Omron CX-Programmer project NewProject (CX-Programmer 9.32)

# PLC NewPLC1: CP1H XA

## Global symbols (name address type ; comment)
AGITATOR SCP
0.00 BOOL  ; Tablet Countinng Proxy
0.01 BOOL  ; Air pressure
0.02 BOOL  ; Turret Motor Overload
0.03 BOOL  ; LH Feeder Motor Overload
0.04 BOOL  ; LH Tamping
0.05 BOOL  ; RH Dozzer Asembly
0.06 BOOL  ; LH Main Set Pressure
0.07 BOOL  ; RH Tamping
0.08 BOOL  ; Guards Limit Switch
0.09 BOOL  ; LH Dozzer Assembly
0.10 BOOL  ; Std. Lubrication Oil Level Low
0.11 BOOL  ; Hydraulic Pressure S/w
100.00 BOOL  ; Main Motor
100.01 BOOL  ; Agitator Motor
100.02 BOOL  ; LH Feeder Motor
100.03 BOOL  ; RH Feeder Motor
100.04 BOOL  ; Hyd. Motor
100.05 BOOL  ; Sampling Gate
100.06 BOOL  ; Hyd. Dec SOV
100.07 BOOL  ; Magnetic Clutch
101.00 BOOL  ; 1 st Layer Sampling Gate ON
101.01 BOOL  ; 1 st Layer Sampling Gate OFF
101.02 BOOL  ; Lubrication Sol. On
101.03 BOOL  ; Comp. Zone Light
101.04 BOOL  ; Dust Extractor
101.05 BOOL  ; LPSL SOV
101.06 BOOL  ; Sampling Hooter
101.07 BOOL  ; Hooter
102 CHANNEL  ; RH Feeder Speed Reference
106.00 BOOL  ; LH Discharge SOV
106.01 BOOL  ; LH Filteration SOV
106.02 BOOL  ; LH Conveyour SOV
106.03 BOOL  ; RH Discharge SOV
106.04 BOOL  ; RH Filteration SOV
106.05 BOOL  ; RH Conveyour SOV
106.06 BOOL  ; Vacuum Pump
1.00 BOOL  ; RH Main Set Pressure
1.01 BOOL  ; RH Feeder Motor Overload
1.02 BOOL  ; Hyd. Motor O/L
1.03 BOOL  ; Emergency Stop
1.04 BOOL  ; LH Powder Level Low
1.05 BOOL  ; RH Powder Level Low
1.06 BOOL  ; Hyd. Oil Level Low
1.07 BOOL  ; LH Feeder Jamming
1.08 BOOL  ; RH Feeder Jamming
1.09 BOOL  ; Door For Ele. Panel Box
1.10 BOOL  ; Hand Wheel Guard
1.11 BOOL  ; Agitator Motor O/L
200 CHANNEL  ; Spare
201 CHANNEL  ; Turret Motor Current
2012 CHANNEL  ; LH Main Punch Force Input
202 CHANNEL  ; Hyd. System Pressure (4-20mA)
203 CHANNEL  ; Spare
210 CHANNEL  ; Turret Motor Speed Reference
211 CHANNEL  ; LH Feeder RPM Speed Refence
2.00 BOOL  ; LOWER GUARD LH OPEN
2.01 BOOL  ; $?St$Bk?_#[591] / LOWER GUARD RH OPEN / $?St$Bk?_#[591]
2.02 BOOL  ; UPPER GUARD FRONT OPEN
2.03 BOOL  ; UPPER GUARD LH OPEN
2.04 BOOL  ; UPPER GUARD RH OPEN
2.05 BOOL  ; UPPER GUARD REAR OPEN
2.06 BOOL  ; Int. Lub Motor Overload/LH POWDER LEVEL VERY LOW
2.07 BOOL  ; Int. Lub Oil Level Low/RH POWDER LEVEL VERY LOW
3.00 BOOL  ; Vacuum Pump O/L
3.01 BOOL  ; Vacum Pump Run Feedback
3.02 BOOL  ; LH Hopper Level High
3.03 BOOL  ; RH Hopper Level High
3.04 BOOL  ; Phase Failure
60 CHANNEL  ; minutes
A351 CHANNEL  ; MINUTE & SECOND
A352 CHANNEL  ; DATE & HOUR
A353 CHANNEL  ; YEAR & MONTH
C0 CHANNEL  ; Turret RPM Counter
C0001 BOOL  ; Lubrication ON Time
C0002 BOOL  ; Lubrication OFF Time
C0003 BOOL  ; Tablet Counter C3
C0005 BOOL  ; Reject Tab. / Rev.
C0006 BOOL  ; High Rejection For 3 Rot.
C0007 BOOL  ; Punch Tight Counter
C0008 BOOL  ; Counter For Sample
C0009 BOOL  ; Counter For Intermittent Cycle
C0010 BOOL  ; Total Rej. In 1 Batch
C0012 BOOL  ; First Rot. Rej. Counter
C0020 BOOL  ; LPSL ON Time
C0021 BOOL  ; LPSL OFF Time
C0025 BOOL  ; second counting
C0026 BOOL  ; minute counting
C0027 BOOL  ; hour counting
C0030 BOOL  ; Sampling interval timer
C0031 BOOL  ; 5 Min delay for machine stop
C0051 BOOL  ; LH Level High CNT
C0052 BOOL  ; RH Level High CNT
C0053 BOOL  ; LH Discharge CNT
C0054 BOOL  ; LH Delay CNT
C0055 BOOL  ; LH Filteration CNT
C0056 BOOL  ; LH Conv CNT
C0057 BOOL  ; RH Discharge CNT
C0058 BOOL  ; RH Delay CNT
C0059 BOOL  ; RH Filteration CNT
C0060 BOOL  ; RH Conv CNT
C11 CHANNEL  ; Total Sample Tab. In 1 Batch
D0 CHANNEL  ; Actual Screen
D1 CHANNEL  ; Operator Password
D1000 CHANNEL  ; Total Tablet Produced LSB
D1005 CHANNEL  ; Total Tablet Produced MSB
D101 CHANNEL  ; Actual Turret RPM
D1050 CHANNEL  ; Total Tablet Produced
D109 CHANNEL  ; Total Tablet Produced Higher Bit
D1100 CHANNEL  ; Main Force Data Range 1100-1199
D1110 CHANNEL  ; Actual Batch size
D1114 CHANNEL  ; Current Range
D116 CHANNEL  ; Current Factor (Count)
D122 CHANNEL  ; Turret Motor Current
D123 CHANNEL  ; Set Lubrication ON Time (Sec.)
D124 CHANNEL  ; Set Lubrication OFF Time (Min.)
D126 CHANNEL  ; Lubrication OFF Time (Min)
D127 CHANNEL  ; Actual Lub. ON Time
D128 CHANNEL  ; Actual Lub. OFF Time
D130 CHANNEL  ; Time For Punch Force Data
D135 CHANNEL  ; Time for Air Blow
D139 CHANNEL  ; Air Blow Delay Time
D141 CHANNEL  ; Air Blow Time Delay
D142 CHANNEL  ; Tablet Counting C3 Data
D152 CHANNEL  ; Main Force Data
D154 CHANNEL  ; High Rejection Limit
D155 CHANNEL  ; Low Rejection Limit
D156 CHANNEL  ; Main Force Data Count
D157 CHANNEL  ; Total Main Force
D159 CHANNEL  ; M/C Station
D161 CHANNEL  ; Main Avg. Force
D165 CHANNEL  ; Avg. Force For Die Fill PID Control
D173 CHANNEL  ; Punch Force For Graph
D180 CHANNEL  ; Force Rejection For Punch1
D181 CHANNEL  ; Force Rejection For Punch2
D182 CHANNEL  ; Force Rejection For Punch3
D183 CHANNEL  ; Force Rejection For Punch4
D184 CHANNEL  ; Force Rejection For Punch5
D185 CHANNEL  ; Air Blow ON Time
D186 CHANNEL  ; Air Blow ON Time (BCD)
D190 CHANNEL  ; Sample Punch No 1
D191 CHANNEL  ; Sample Punch No 2
D192 CHANNEL  ; Sample Punch No 3
D193 CHANNEL  ; Sample Punch No 4
D194 CHANNEL  ; Sample Punch No 5
D195 CHANNEL  ; Counter/Time Value For Sampling
D198 CHANNEL  ; Sample Time
D2 CHANNEL  ; Manager Password
D200 CHANNEL  ; minutes
D2000 CHANNEL  ; MINUTE & SECOND
D2002 CHANNEL  ; SEC
D2003 CHANNEL  ; MIN
D201 CHANNEL  ; hours
D2012 CHANNEL  ; HOUR
D2013 CHANNEL  ; DATE
D2022 CHANNEL  ; MONTH
D2023 CHANNEL  ; YEAR
D21 CHANNEL  ; Password for Login
D22 CHANNEL  ; Operator Password
D226 CHANNEL  ; Time Interval for Sampling (Sec)
D23 CHANNEL  ; Supervisor Password
D230 CHANNEL  ; Sampling Gate ON Time
D232 CHANNEL  ; Time For Intermittent Cycle
D236 CHANNEL  ; Total Rej. In 1 Batch
D238 CHANNEL  ; Total Sample Tab. In 1 Batch
D24 CHANNEL  ; Manager Password
D241 CHANNEL  ; High Force Control Limit
D242 CHANNEL  ; Low Force Control Limit
D243 CHANNEL  ; Initial Rejection Tablet
D245 CHANNEL  ; Enter Sync. Percentage
D25 CHANNEL  ; Selection Change Password
D250 CHANNEL  ; Vac-U-Max Control
D252 CHANNEL  ; (Set Turret RPM-Min RPM)
D254 CHANNEL  ; LH Delay Time
D256 CHANNEL  ; LH Filteration Time
D258 CHANNEL  ; Set Main Pressure
D26 CHANNEL  ; Enter Old Password
D260 CHANNEL  ; Set Tamping Pressure
D261 CHANNEL  ; Set Depth of Die Fill
D262 CHANNEL  ; Set Main Tablet Thickness
D264 CHANNEL  ; Set Tamp. Tab. Thickness
D266 CHANNEL  ; Actual Depth of Die Fill
D268 CHANNEL  ; Actual Tablet Thickness
D27 CHANNEL  ; Enter New Password
D270 CHANNEL  ; Actual Tamping Tablet Thickness
D272 CHANNEL  ; Main Upper Punch Entry
D274 CHANNEL  ; Tamping Upper Punch Entry
D275 CHANNEL  ; Message For Sampling collection
D276 CHANNEL  ; Die Fill Position message
D277 CHANNEL  ; Tablet Thickness Message
D278 CHANNEL  ; Tamp. Tablet Thickness Message
D28 CHANNEL  ; 0=Enter Password 1= Password OK 2=Invalid Password
D280 CHANNEL  ; RH Dischrge Time (BCD)
D286 CHANNEL  ; Tamping Force Data
D288 CHANNEL  ; LH High Level Disappear Time (BCD)
D29 CHANNEL  ; Change Password Message
D290 CHANNEL  ; RH High Level Disappear Time (BCD)
D296 CHANNEL  ; Total Cycle
D298 CHANNEL  ; Total Cycle (BCD)
D30 CHANNEL  ; RH Feeder RPM
D300 CHANNEL  ; RH Feeder RPM
D3015 CHANNEL  ; LH scp input min
D3016 CHANNEL  ; LH scp scal min
D3017 CHANNEL  ; LH scp scal max
D3018 CHANNEL  ; LH scp input max
D3019 CHANNEL  ; Actual LH Punch Force
D302 CHANNEL  ; Hour
D304 CHANNEL  ; Min
D306 CHANNEL  ; Sec
D319 CHANNEL  ; RH Store Feeder RPM
D330 CHANNEL  ; Sampling inteval time min
D3508 CHANNEL  ; Operator Code
D3509 CHANNEL  ; Recipe Code
D3525 CHANNEL  ; Batch Size
D360 CHANNEL  ; Tamp. Avg Force
D364 CHANNEL  ; Tamping Trend Graph
D368 CHANNEL  ; Avg. Ejection Data
D39 CHANNEL  ; RH Store Feeder RPM
D40 CHANNEL  ; Store Screen
D4000 CHANNEL  ; minutes
D4001 CHANNEL  ; hours
D406 CHANNEL  ; Ejection Force Data
D432 CHANNEL  ; Die Fill MIN
D433 CHANNEL  ; Die Fill MAX
D435 CHANNEL  ; Machine Station
D44 CHANNEL  ; Set Turret RPM (Store)
D480 CHANNEL  ; Acceleration
D481 CHANNEL  ; Deacceleration
D482 CHANNEL  ; Frequency
D484 CHANNEL  ; Pulses
D486 CHANNEL  ; Start Frequency
D499 CHANNEL  ; Main Lower Punch Position
D500 CHANNEL  ; Tamping interlock
D501 CHANNEL  ; Main Pressure Interlock
D510 CHANNEL  ; Set LPSL ON Time
D511 CHANNEL  ; Set LPSL OFF Time
D512 CHANNEL  ; LPSL ON TIME (Sec)
D513 CHANNEL  ; LPSL OFF TIME (Min)
D514 CHANNEL  ; Output Pulse to be Generate
D515 CHANNEL  ; Act. LPSL ON Time
D516 CHANNEL  ; Act. LPSL OFF Time
D52 CHANNEL  ; LH Set Feeder RPM
D520 CHANNEL  ; Hyd. Low Limit
D521 CHANNEL  ; Hyd. High Limit
D522 CHANNEL  ; Hyd. Limit Low (Comp)
D523 CHANNEL  ; Hyd. Limit High (Comp)
D525 CHANNEL  ; Hyd. Sys. Pr. Message
D527 CHANNEL  ; Act. Hyd. Pressure
D528 CHANNEL  ; Hyd. Graph
D53 CHANNEL  ; LH Store Feeder RPM
D530 CHANNEL  ; SCL_P
D533 CHANNEL  ; SCL_P3
D535 CHANNEL  ; Total travel in mm/100
D539 CHANNEL  ; Tamping Lower Punch Position
D54 CHANNEL  ; LH Store Feeder RPM
D542 CHANNEL  ; Total Cup Depth
D548 CHANNEL  ; Lower punch pos + Total Cup Depth
D550 CHANNEL  ; Set Agitator RPM
D552 CHANNEL  ; Act Agitiator RPM
D56 CHANNEL  ; Feeder RPM (Float)
D572 CHANNEL  ; Time Interval For Sampling (BCD) - Sec
D578 CHANNEL  ; Die Fill High+Low Limit
D579 CHANNEL  ; Die Fill High/Low Avg Limit
D60 CHANNEL  ; RH Feeder O/P
D601 CHANNEL  ; Set Main  + Relief
D602 CHANNEL  ; Set Tamping + Relief Value
D606 CHANNEL  ; No of Tablet Counter
D615 CHANNEL  ; Min. Main Force
D6150 CHANNEL  ; -
D6152 CHANNEL  ; Total Rejec.+Sample Tab
D6158 CHANNEL  ; Powder Delay Time
D6160 CHANNEL  ; M/c Stn (Print)
D6168 CHANNEL  ; Feeder Post Run Time (BCD)
D617 CHANNEL  ; Max. Main Force
D619 CHANNEL  ; Min. Tamp. Force
D621 CHANNEL  ; Max. Tamp. Force
D64 CHANNEL  ; Scale Min
D66 CHANNEL  ; Scale Range
D67 CHANNEL  ; \
D7 CHANNEL  ; '
D70 CHANNEL  ; Die Fill Position
D700 CHANNEL  ; Lower Punch position at last time
D7005 CHANNEL  ; Batch Size
D702 CHANNEL  ; Store lower punch Position at last time
D7050 CHANNEL  ; Hour
D7052 CHANNEL  ; Min
D7060 CHANNEL  ; Sample + Reject Tab
D7064 CHANNEL  ; Good Tablet
D707 CHANNEL  ; Generate Pulse at last time
D709 CHANNEL  ; Total Travel at last time
D710 CHANNEL  ; Required pulse for travel at last time
D712 CHANNEL  ; Overl pulse at last time
D715 CHANNEL  ; Pulse feedback
D720 CHANNEL  ; Every 0.2 sec Set Tamp. Tab Thickness
D74 CHANNEL  ; LH Actual Feeder RPM
D746 CHANNEL  ; Powder Feeding Selection
D747 CHANNEL  ; Hour Meter 0:Reset 1:Start
D748 CHANNEL  ; Guard Interlock
D749 CHANNEL  ; Dummy Selection
D75 CHANNEL  ; Set Turret RPM
D750 CHANNEL  ; Dummy 1
D751 CHANNEL  ; Dummy 2
D752 CHANNEL  ; Dummy 3
D753 CHANNEL  ; Dummy 4
D754 CHANNEL  ; Dummy 5
D756 CHANNEL  ; Mode of Sampling
D758 CHANNEL  ; Compaction Mode 0: Manual 1: Auto
D759 CHANNEL  ; SCADA_BYPASS
D76 CHANNEL  ; Store Turret RPM
D762 CHANNEL  ; Dummy Punch Count
D764 CHANNEL  ; Total Dummy Punch
D766 CHANNEL  ; Final Total Punch
D768 CHANNEL  ; Tab w Dummy Punch
D77 CHANNEL  ; RH Actual Feeder RPM
D78 CHANNEL  ; RPM (Float)
D8 CHANNEL  ; Change Screen
D800 CHANNEL  ; Act. Hyd. Pressure Print
D82 CHANNEL  ; Input Max
D86 CHANNEL  ; Scale Min
D88 CHANNEL  ; Scale Range
D96 CHANNEL  ; Used for Turret RPM Calculation
D99 CHANNEL  ; Total No. Of Punch
H100.00 BOOL  ; Dummy Punch Selection
H100.01 BOOL  ; 0: Gravity 1: Force Feeder
H100.02 BOOL  ; Sampling ON/OFF
H100.03 BOOL  ; Batch Reseted
H101 CHANNEL  ; Hydrualic Pressure
H101.00 BOOL  ; Lub, Healthy
H102 CHANNEL  ; Hydraulic Pressure for Graph
H102.00 BOOL  ; LPSL ON Time : Low Limit
H102.01 BOOL  ; LPSL ON Time : Upper Limit
H102.02 BOOL  ; LPSL OFF Time : Low Limit
H102.03 BOOL  ; LPSL OFF Time : Upper Limit
H102.04 BOOL  ; LPSL Healthy
H102.05 BOOL  ; 1 Min Pulse
H103 CHANNEL  ; Turret Motor Current * 10
H103.00 BOOL  ; System Pr. High IL
H103.01 BOOL  ; Sys. Pr. Low IL
H103.02 BOOL  ; Hyd. Sys. Pr. High
H103.03 BOOL  ; Hyd. Sys. Pr. Low
H103.05 BOOL  ; 0: Hyd. Manual 1: Hyd. Auto
H103.06 BOOL  ; Hyd. Healthy
H103.07 BOOL  ; Hyd. INC
H103.08 BOOL  ; Hyd. DEC
H103.15 BOOL  ; All Upper Punch Free
H105.00 BOOL  ; Scada 0: OFF 1:Running
H105.01 BOOL  ; Scada 0: Bypass 1: Interlock
H107 CHANNEL  ; Actual Tab/Min
H10.00 BOOL  ; Bilayer sel. 1: standard 0: Bilayer
H10.01 BOOL  ; Bilayer Sampling
H10.02 BOOL  ; Calibration bit for current in calibration screen
H10.04 BOOL  ; Bilayer Sampling ON
H10.05 BOOL  ; Bilayer sampled on
H110.00 BOOL  ; Punch Tight 1
H110.01 BOOL  ; Punch Tight 2
H110.02 BOOL  ; Punch Tight 3
H110.03 BOOL  ; Punch Tight 4
H110.04 BOOL  ; Punch Tight 5
H110.05 BOOL  ; Punch Tight 6
H110.06 BOOL  ; Punch Tight 7
H110.07 BOOL  ; Punch Tight 8
H110.08 BOOL  ; Punch Tight 9
H110.09 BOOL  ; Punch Tight 10
H110.10 BOOL  ; Punch Tight 11
H110.11 BOOL  ; Punch Tight 12
H110.12 BOOL  ; Punch Tight 13
H110.13 BOOL  ; Punch Tight 14
H110.14 BOOL  ; Punch Tight 15
H110.15 BOOL  ; Punch Tight 16
H111.00 BOOL  ; Punch Tight 17
H111.01 BOOL  ; Punch Tight 18
H111.02 BOOL  ; Punch Tight 19
H111.03 BOOL  ; Punch Tight 20
H111.04 BOOL  ; Punch Tight 21
H111.05 BOOL  ; Punch Tight 22
H111.06 BOOL  ; Punch Tight 23
H111.07 BOOL  ; Punch Tight 24
H111.08 BOOL  ; Punch Tight 25
H111.09 BOOL  ; Punch Tight 26
H111.10 BOOL  ; Punch Tight 27
H111.11 BOOL  ; Punch Tight 28
H111.12 BOOL  ; Punch Tight 29
H111.13 BOOL  ; Punch Tight 30
H111.14 BOOL  ; Punch Tight 31
H111.15 BOOL  ; Punch Tight 32
H112.00 BOOL  ; Punch Tight 33
H112.01 BOOL  ; Punch Tight 34
H112.02 BOOL  ; Punch Tight 35
H112.03 BOOL  ; Punch Tight 36
H112.04 BOOL  ; Punch Tight 37
H118 CHANNEL  ; Actual Turret RPM
H11.00 BOOL  ; Download Recipe
H11.01 BOOL  ; Bilayer Sampling latch bit
H123 CHANNEL  ; Batch Recipe Code
H12.14 BOOL  ; Screen Move for MS1
H12.15 BOOL  ; Screen Move for MS2
H140.00 BOOL  ; Agitator Jog
H140.01 BOOL  ; Agitator ON/OFF
H150 CHANNEL  ; Total Tablet Produced Lower Bit
H150.01 BOOL  ; View Recipe
H150.02 BOOL  ; Download Recipe
H150.03 BOOL  ; Batch Print
H150.04 BOOL  ; Batch Print ON
H150.05 BOOL  ; Batch Start (Once)
H151.00 BOOL  ; MS1 Screen
H151.01 BOOL  ; MS2 SCREEN
H151.02 BOOL  ; Auto Return From MS1
H151.03 BOOL  ; Return
H151.04 BOOL  ; Auto Return From MS2
H151.05 BOOL  ; Auto Return From MS3
H151.06 BOOL  ; MS3 screen
H151.07 BOOL  ; MS4 screen
H151.08 BOOL  ; Auto Return From MS4
H16.00 BOOL  ; Sampling Alarm Time cycle Latch
H16.01 BOOL  ; Sampling timer Done
H16.02 BOOL  ; 5 Min delay timer done
H16.04 BOOL  ; Hooter on
H17.00 BOOL  ; Interlock for Sampling time Inc
H17.01 BOOL  ; Interlock for Sampling time Dec
H18.00 BOOL  ; Dust Ext. Start
H18.01 BOOL  ; Dust Ext. Stop
H18.02 BOOL  ; Dust Ext. On
H21.00 BOOL  ; Operator
H21.01 BOOL  ; Supervisor
H21.02 BOOL  ; Manager
H21.08 BOOL  ; Supervisor / Manger Login
H21.09 BOOL  ; Operator Password OK
H21.10 BOOL  ; Supervisor Password OK
H21.11 BOOL  ; Manager Password OK
H21.12 BOOL  ; Password OK
H222.00 BOOL  ; Batch Complete Latch
H22.00 BOOL  ; Operator Old Password OK
H22.01 BOOL  ; Supervisor Old Password OK
H22.02 BOOL  ; Manager Old Password OK
H22.03 BOOL  ; Old Password OK
H22.05 BOOL  ; Security Control Bit
H22.06 BOOL  ; Master Password Bit
H22.07 BOOL  ; Operator Once Bit
H22.08 BOOL  ; Supervisor Once Bit
H22.09 BOOL  ; Manager Once Bit
H22.12 BOOL  ; Change Operator Password
H22.13 BOOL  ; Change Supervisor Password
H22.14 BOOL  ; Change Manager Password
H23.01 BOOL  ; Change Operator Password Once Bit
H23.03 BOOL  ; Change Supervisor Password Once Bit
H23.05 BOOL  ; Change Manager Password Once Bit
H25.01 BOOL  ; Air Pressure Set
H25.07 BOOL  ; Int Lub oil Level Low Latch
H25.10 BOOL  ; Lubrication Oil Level Low Set
H25.11 BOOL  ; Hydraulic Pressure S/w Set
H26.06 BOOL  ; Hyd. Oil Level Low Set
H36.00 BOOL  ; Vac-U-Max Reset
H36.01 BOOL  ; Vac-U-Max Start/Stop
H36.02 BOOL  ; Vac-U-Max Hault
H36.05 BOOL  ; Vac-U-Max Healthy Auto
H36.06 BOOL  ; LH Vac-U-Max Running
H36.07 BOOL  ; RH Vac-U-Max Running
H36.08 BOOL  ; Total Cycle Complete
H36.09 BOOL  ; LH Hopper Level High (Latch)
H36.10 BOOL  ; RH Hopper Level High (Latch)
H387 CHANNEL  ; h120
H400.00 BOOL  ; Hooter Reset
H400.05 BOOL  ; Hooter latch
H50.00 BOOL  ; VAC U MAX 0=man 1=auto
H50.01 BOOL  ; LH Discharge SOV ON/OFF
H50.02 BOOL  ; LH Filteration SOV ON/OFF
H50.03 BOOL  ; LH Conveyour SOV ON/OFF
H50.04 BOOL  ; RH Discharge SOV ON/OFF
H50.05 BOOL  ; RH Filteration SOV ON/OFF
H50.06 BOOL  ; RH Conveyour SOV ON/OFF
H50.07 BOOL  ; Vacuum Pump ON/OFF
H51.00 BOOL  ; Main Interlock Healthy
H51.01 BOOL  ; Main Motor Start
H51.02 BOOL  ; Main Motor RUN (Auto)
H51.03 BOOL  ; Main Motor Stop
H51.04 BOOL  ; Lubrication Jog
H51.05 BOOL  ; Turret & Feeder Jog
H51.06 BOOL  ; Clutch Engage
H51.07 BOOL  ; Clutch Latch
H51.08 BOOL  ; 0=Gurds Bypass 1=Guards Interlock
H51.09 BOOL  ; Clutch Disengage
H51.10 BOOL  ; 0=Manual 1=Auto
H51.11 BOOL  ; Lub.: 0=Auto 1= Manual
H51.12 BOOL  ; Turret Jog
H51.13 BOOL  ; LH Feeder Motor Jog
H51.14 BOOL  ; RH Feeder Motor Jog
H51.15 BOOL  ; Hydraulic Pressure Dec.
H52.01 BOOL  ; Rising Edge of Proxy
H52.04 BOOL  ; Interlock for Turret RPM Inc
H52.05 BOOL  ; Interlock for Turret RPM Dec
H52.06 BOOL  ; LH Interlock for Feeder RPM Inc
H52.07 BOOL  ; LH Interlock for Feeder RPM Dec
H52.08 BOOL  ; RH Interlock for Feeder RPM Inc
H52.09 BOOL  ; RH Interlock for Feeder RPM Dec
H52.10 BOOL  ; Main Motor (Test RUN)
H52.11 BOOL  ; LPSL 0: Manual 1: Auto
H52.12 BOOL  ; Initial Rej. Gate Dignostic
H52.13 BOOL  ; LPSL Jog
H53.00 BOOL  ; Batch Complete
H53.01 BOOL  ; Batch Reset
H53.02 BOOL  ; Lower Limit Lubrication ON Time
H53.03 BOOL  ; Upper Limit Lubrication ON Time
H53.04 BOOL  ; Lower Limit Lubrication OFF Time
H53.05 BOOL  ; Upper Limit Lubrication OFF Time
H53.07 BOOL  ; Interlock for Download
H53.07 BOOL  ; Access Denied
H53.08 BOOL  ; Print Command to Scada
H53.09 BOOL  ; Home Proxy not Proper
H53.10 BOOL  ; Tablet Count Proxy Not Proper
H53.12 BOOL  ; Die Fill at Min Limit
H53.13 BOOL  ; Die Fill at Max Limit
H54.00 BOOL  ; Selected Punch
H54.01 BOOL  ; All Tab. Continuous
H54.02 BOOL  ; All Tablet Intermittent
H54.03 BOOL  ; Dynemic Reject on
H54.04 BOOL  ; For 1 Rot. High Rejection
H54.05 BOOL  ; Tablet Rejection/Rev.
H54.06 BOOL  ; Counter NEQ Zero
H54.07 BOOL  ; No. of Tablet
H54.08 BOOL  ; Stop Reason Latch
H54.09 BOOL  ; Final Bit For Rej./Samp.
H54.10 BOOL  ; Air Blow ON Time Bit
H54.11 BOOL  ; Sample Enable For 1 Rot.
H54.12 BOOL  ; Rej. Air Blow On Dignostic
H54.13 BOOL  ; $?St$Bk?_#[592] / 0=Rotation 1=Time / (Now only Based on Time)$?St$Bk?_#[592]
H54.14 BOOL  ; 0=Sample OFF 1=Sample On
H54.15 BOOL  ; All Tablet Intermittent
H55 CHANNEL  ; Interlock Status
H55.00 BOOL  ; For Input Interlocks
H56 CHANNEL  ; Interlock Status
H56.00 BOOL  ; For Input Interlocks
H56 CHANNEL  ; Interlock Status
H57 CHANNEL  ; Interlock Status
H57.02 BOOL  ; LH POWDER VACCUM HOPPER
H57.03 BOOL  ; RH POWDER VACCUM HOPPER
H58.00 BOOL  ; Pop up for Access Denied
H59.01 BOOL  ; Sampleing Enable Bit
H59.02 BOOL  ; Reset for C8
H59.03 BOOL  ; Reset For C8 & C9
H59.04 BOOL  ; Complete Intermittent Cycle
H60.01 BOOL  ; Rejection/Sampling For Perticular Punch
H61.01 BOOL  ; Tab. For Sampling
H62.00 BOOL  ; 0=Sync. Manual 1=Sync. Auto
H62.01 BOOL  ; Main Pressure O/L
H62.02 BOOL  ; Tamping Pressure O/L
H62.03 BOOL  ; 0=Die Fill Manual 1= Diefill Auto
H62.04 BOOL  ; Die Fill  Maximum
H62.05 BOOL  ; Die Fill Minimum
H62.06 BOOL  ; Tablet Thickness Maximum
H62.07 BOOL  ; Tablet Thickness Minimum
H62.08 BOOL  ; Tamp. Tab. Thickness Maximum
H62.09 BOOL  ; Tamp. Tab. Thickness Minimum
H63.04 BOOL  ; Batch Start for Scada
H63.05 BOOL  ; Batch Complete for Scada
H64.00 BOOL  ; Avg Force < Lower Force Limit
H64.02 BOOL  ; Avg Force > Upper Force Limit
H64.04 BOOL  ; Die Fill Inc
H64.05 BOOL  ; Die Fill Dec
H64.06 BOOL  ; Die Fill INC (HMI)
H64.07 BOOL  ; Die Fill DEC (HMI)
H64.08 BOOL  ; Tamp. Tab Thickness Inc
H64.09 BOOL  ; Tamp. Tab. Thickness Dec.
H65.00 BOOL  ; Output Interlocks
H66.00 BOOL  ; Output Interlocks
H67.00 BOOL  ; Output Interlocks
H68.00 BOOL  ; Tamping Tablet Thickness Sevo Interlock
H68.01 BOOL  ; Tamping Servo REV at last time
H68.02 BOOL  ; Tamping servo FWD at Last time
H70.00 BOOL  ; 1 sec pulse o/p latch
H70.03 BOOL  ; All Tab. Cont.
H70.05 BOOL  ; No. of. Tab. Enb.
H70.07 BOOL  ; Ejection Force Limit Max
H70.10 BOOL  ; Batch No Enter
H72.05 BOOL  ; Vac U Max Healthy Man
H75.02 BOOL  ; Station 20
H75.03 BOOL  ; Station 24
H75.04 BOOL  ; Station 30
H77.00 BOOL  ; Agitator Interlock/Bypass
H77.14 BOOL  ; Reset all counter for RH & count 1 cycle
H77.15 BOOL  ; Reset all counter for LH & count 1 cycle
H7.01 BOOL  ; Manual Interlock
H7.02 BOOL  ; Test Turret Interlock
H7.03 BOOL  ; Test LH Feeder Interlock
H7.04 BOOL  ; Test RH Feeder Interlock
H7.05 BOOL  ; Test Air Interlock
H7.06 BOOL  ; Feeder Jaming 0: Bypass 1: Interlock
H7.07 BOOL  ; LH Feeder Jamming Interlock
H7.08 BOOL  ; RH Feeder Jamming Interlock
H80.00 BOOL  ; 0:Two Side,1:Single side
T0007 BOOL  ; Hyd. Dec SOV OFF Time
T0013 BOOL  ; LH Feeder Jamming Timer
T0018 BOOL  ; Sampling Gate ON Timer
T0023 BOOL  ; Clutch Engage (Aft Feeder Pre Run)
T0024 BOOL  ; Actual Pusle for every 10 Sec
T0025 BOOL  ; Clutch Delay (Auto)
T0028 BOOL  ; Feeder Post Run Timer
T0029 BOOL  ; Powder Level Timer
T0034 BOOL  ; LH Feeder RPM Actual Transfer Time
T0035 BOOL  ; Lubrication Automatically Auto after 5 Min.
T0036 BOOL  ; Access Denied Timer (1s)
T0037 BOOL  ; RH Feeder RPM Actual Transfer Time
HYD_PRESSURE SCP
Hyd_New SCP_Hyd
LH_FEEDER_SPEED SCP
RH_Feeder_Reference SCP
RTC_01 FRTC
Turret_Current SCP
Turret_Speed_reference SCP

## Program Main_Program (cyclic task 0)
Local symbols
AD0 CHANNEL
D441D454 CHANNEL
D441d454 CHANNEL
D442D452 CHANNEL
D444D454 CHANNEL
D4d425 INT
DD411 INT
Dd568 INT
Dd572 UINT_BCD
Dh102 INT
First_pass BOOL
P_0_01s BOOL
P_on BOOL  ; Always on flag
cf CHANNEL
cfg CHANNEL
ch0 CHANNEL
cio2 INT
cntr35 BOOL
ct4 BOOL
d INT
da CHANNEL
dx30 CHANNEL
end BOOL
h BOOL
ld700 UINT
out BOOL
p BOOL
p102 BOOL
p_1s BOOL  ; pulse for 1sec
p_ON BOOL
p_On BOOL
p_oFF BOOL
p_oN BOOL
p_on BOOL  ; always on flag
scl BOOL  ; d200
up BOOL
vw0 CHANNEL

### Section Password
; Pass Word

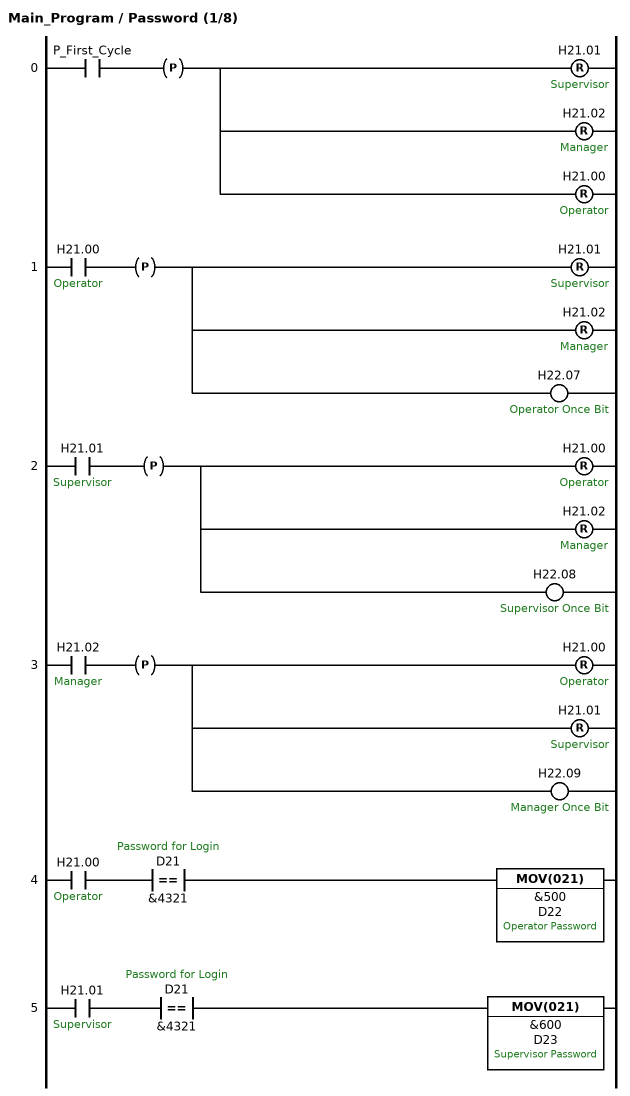
; rung 0
LD P_First_Cycle
UP(521)
RSET H21.01  ; Supervisor
RSET H21.02  ; Manager
RSET H21.00  ; Operator
; rung 1
LD H21.00  ; Operator
UP(521)
RSET H21.01  ; Supervisor
RSET H21.02  ; Manager
OUT H22.07  ; Operator Once Bit
; rung 2
LD H21.01  ; Supervisor
UP(521)
RSET H21.00  ; Operator
RSET H21.02  ; Manager
OUT H22.08  ; Supervisor Once Bit
; rung 3
LD H21.02  ; Manager
UP(521)
RSET H21.00  ; Operator
RSET H21.01  ; Supervisor
OUT H22.09  ; Manager Once Bit
; rung 4
LD H21.00  ; Operator
AND=(300) D21 &4321  ; Password for Login
MOV(021) &500 D22  ; Operator Password
; rung 5
LD H21.01  ; Supervisor
AND=(300) D21 &4321  ; Password for Login
MOV(021) &600 D23  ; Supervisor Password

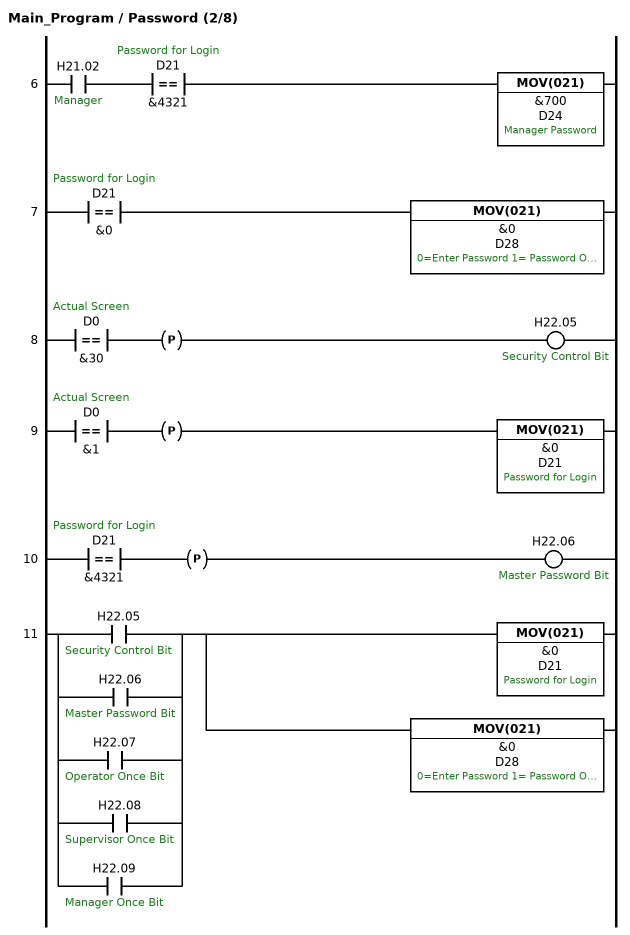
; rung 6
LD H21.02  ; Manager
AND=(300) D21 &4321  ; Password for Login
MOV(021) &700 D24  ; Manager Password
; rung 7
LD=(300) D21 &0  ; Password for Login
MOV(021) &0 D28  ; 0=Enter Password 1= Password OK 2=Invalid Password
; rung 8
LD=(300) D0 &30  ; Actual Screen
UP(521)
OUT H22.05  ; Security Control Bit
; rung 9
LD=(300) D0 &1  ; Actual Screen
UP(521)
MOV(021) &0 D21  ; Password for Login
; rung 10
LD=(300) D21 &4321  ; Password for Login
UP(521)
OUT H22.06  ; Master Password Bit
; rung 11
LD H22.05  ; Security Control Bit
OR H22.06  ; Master Password Bit
OR H22.07  ; Operator Once Bit
OR H22.08  ; Supervisor Once Bit
OR H22.09  ; Manager Once Bit
MOV(021) &0 D21  ; Password for Login
MOV(021) &0 D28  ; 0=Enter Password 1= Password OK 2=Invalid Password

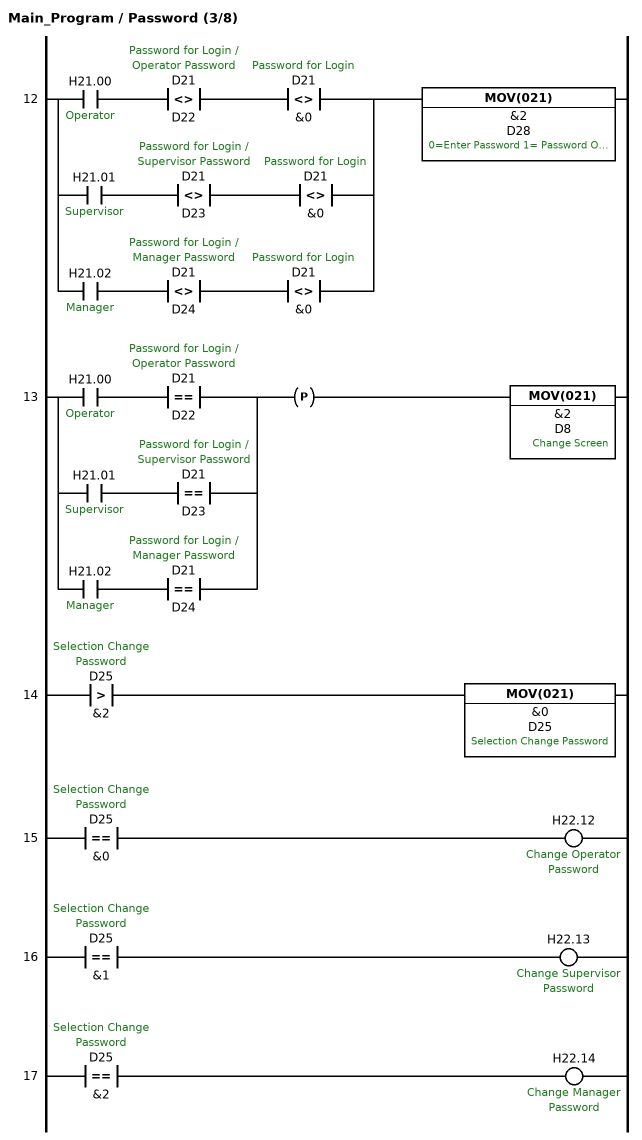
; rung 12
LD H21.00  ; Operator
AND<>(305) D21 D22  ; Password for Login, Operator Password
AND<>(305) D21 &0  ; Password for Login
LD H21.01  ; Supervisor
AND<>(305) D21 D23  ; Password for Login, Supervisor Password
AND<>(305) D21 &0  ; Password for Login
ORLD
LD H21.02  ; Manager
AND<>(305) D21 D24  ; Password for Login, Manager Password
AND<>(305) D21 &0  ; Password for Login
ORLD
MOV(021) &2 D28  ; 0=Enter Password 1= Password OK 2=Invalid Password
; rung 13
LD H21.00  ; Operator
AND=(300) D21 D22  ; Password for Login, Operator Password
LD H21.01  ; Supervisor
AND=(300) D21 D23  ; Password for Login, Supervisor Password
ORLD
LD H21.02  ; Manager
AND=(300) D21 D24  ; Password for Login, Manager Password
ORLD
UP(521)
MOV(021) &2 D8  ; Change Screen
; rung 14
LD>(320) D25 &2  ; Selection Change Password
MOV(021) &0 D25  ; Selection Change Password
; rung 15
LD=(300) D25 &0  ; Selection Change Password
OUT H22.12  ; Change Operator Password
; rung 16
LD=(300) D25 &1  ; Selection Change Password
OUT H22.13  ; Change Supervisor Password
; rung 17
LD=(300) D25 &2  ; Selection Change Password
OUT H22.14  ; Change Manager Password

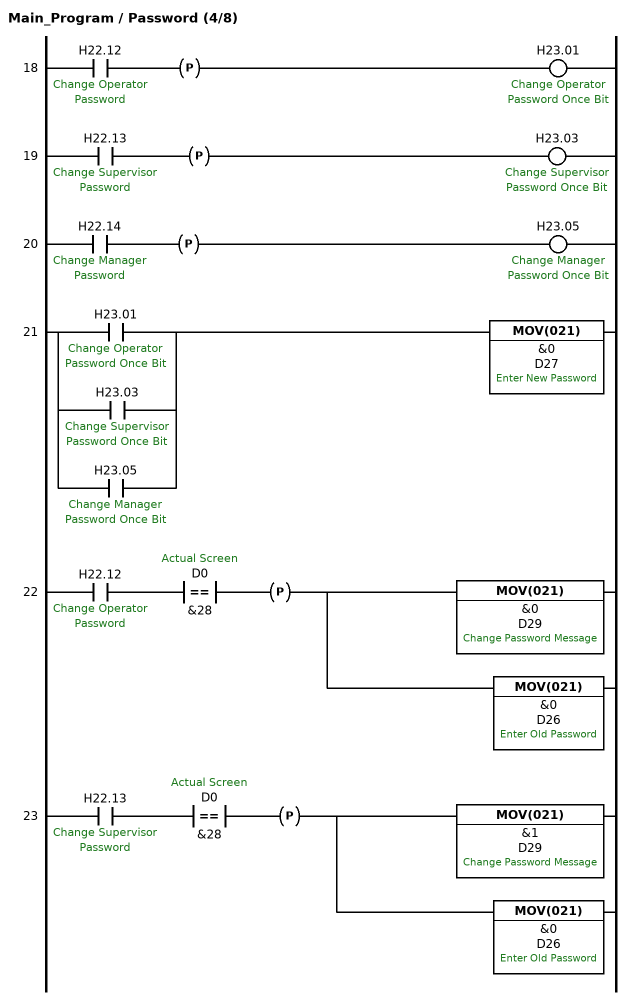
; rung 18
LD H22.12  ; Change Operator Password
UP(521)
OUT H23.01  ; Change Operator Password Once Bit
; rung 19
LD H22.13  ; Change Supervisor Password
UP(521)
OUT H23.03  ; Change Supervisor Password Once Bit
; rung 20
LD H22.14  ; Change Manager Password
UP(521)
OUT H23.05  ; Change Manager Password Once Bit
; rung 21
LD H23.01  ; Change Operator Password Once Bit
OR H23.03  ; Change Supervisor Password Once Bit
OR H23.05  ; Change Manager Password Once Bit
MOV(021) &0 D27  ; Enter New Password
; rung 22
LD H22.12  ; Change Operator Password
AND=(300) D0 &28  ; Actual Screen
UP(521)
MOV(021) &0 D29  ; Change Password Message
MOV(021) &0 D26  ; Enter Old Password
; rung 23
LD H22.13  ; Change Supervisor Password
AND=(300) D0 &28  ; Actual Screen
UP(521)
MOV(021) &1 D29  ; Change Password Message
MOV(021) &0 D26  ; Enter Old Password

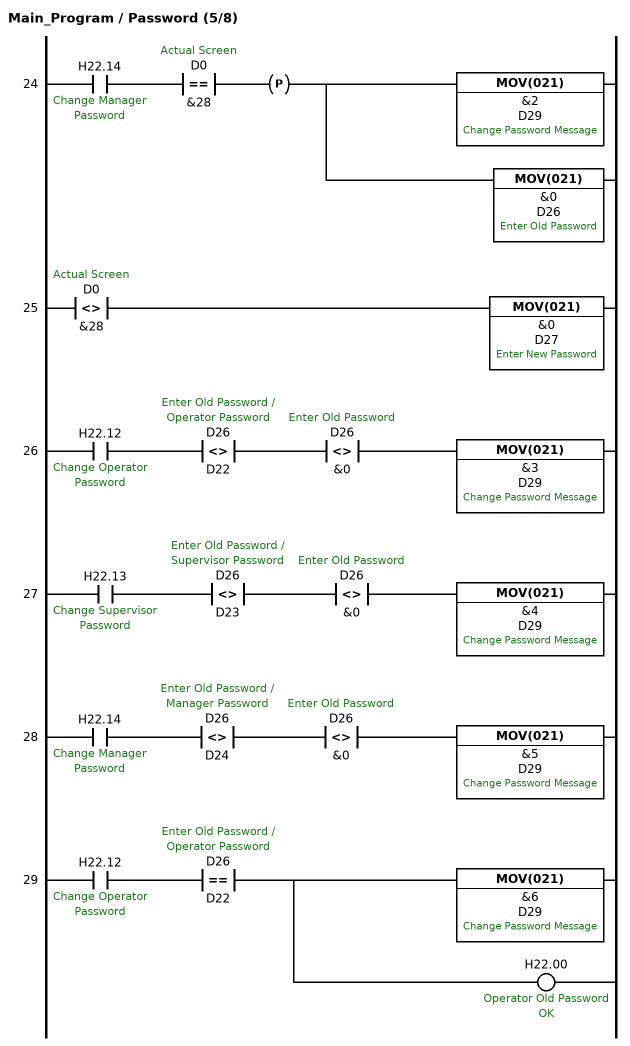
; rung 24
LD H22.14  ; Change Manager Password
AND=(300) D0 &28  ; Actual Screen
UP(521)
MOV(021) &2 D29  ; Change Password Message
MOV(021) &0 D26  ; Enter Old Password
; rung 25
LD<>(305) D0 &28  ; Actual Screen
MOV(021) &0 D27  ; Enter New Password
; rung 26
LD H22.12  ; Change Operator Password
AND<>(305) D26 D22  ; Enter Old Password, Operator Password
AND<>(305) D26 &0  ; Enter Old Password
MOV(021) &3 D29  ; Change Password Message
; rung 27
LD H22.13  ; Change Supervisor Password
AND<>(305) D26 D23  ; Enter Old Password, Supervisor Password
AND<>(305) D26 &0  ; Enter Old Password
MOV(021) &4 D29  ; Change Password Message
; rung 28
LD H22.14  ; Change Manager Password
AND<>(305) D26 D24  ; Enter Old Password, Manager Password
AND<>(305) D26 &0  ; Enter Old Password
MOV(021) &5 D29  ; Change Password Message
; rung 29
LD H22.12  ; Change Operator Password
AND=(300) D26 D22  ; Enter Old Password, Operator Password
MOV(021) &6 D29  ; Change Password Message
OUT H22.00  ; Operator Old Password OK

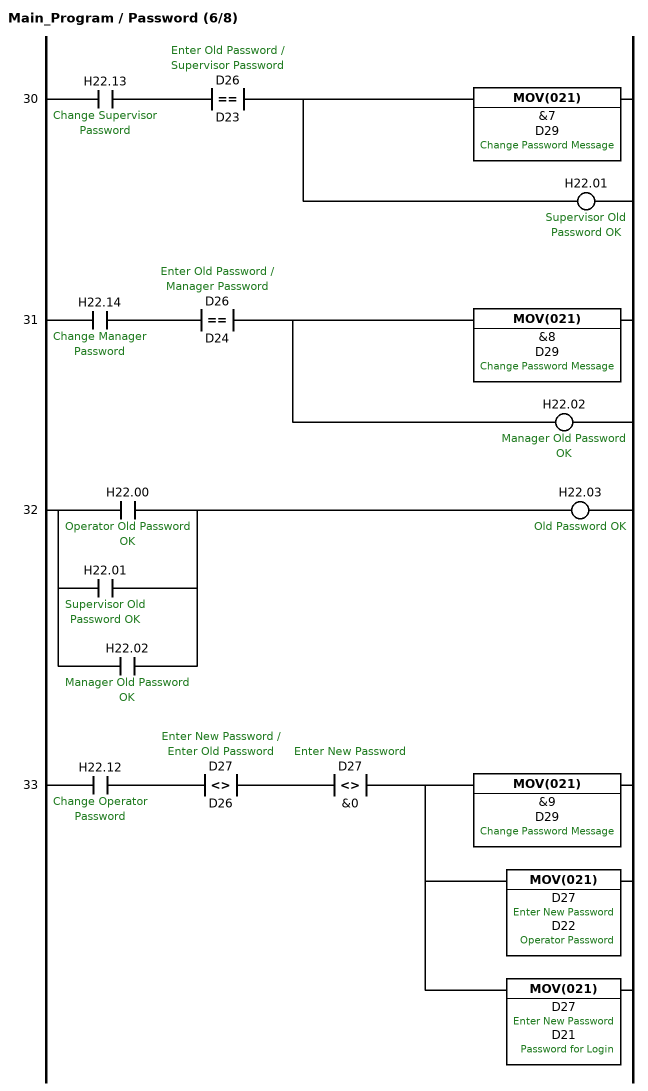
; rung 30
LD H22.13  ; Change Supervisor Password
AND=(300) D26 D23  ; Enter Old Password, Supervisor Password
MOV(021) &7 D29  ; Change Password Message
OUT H22.01  ; Supervisor Old Password OK
; rung 31
LD H22.14  ; Change Manager Password
AND=(300) D26 D24  ; Enter Old Password, Manager Password
MOV(021) &8 D29  ; Change Password Message
OUT H22.02  ; Manager Old Password OK
; rung 32
LD H22.00  ; Operator Old Password OK
OR H22.01  ; Supervisor Old Password OK
OR H22.02  ; Manager Old Password OK
OUT H22.03  ; Old Password OK
; rung 33
LD H22.12  ; Change Operator Password
AND<>(305) D27 D26  ; Enter New Password, Enter Old Password
AND<>(305) D27 &0  ; Enter New Password
MOV(021) &9 D29  ; Change Password Message
MOV(021) D27 D22  ; Enter New Password, Operator Password
MOV(021) D27 D21  ; Enter New Password, Password for Login

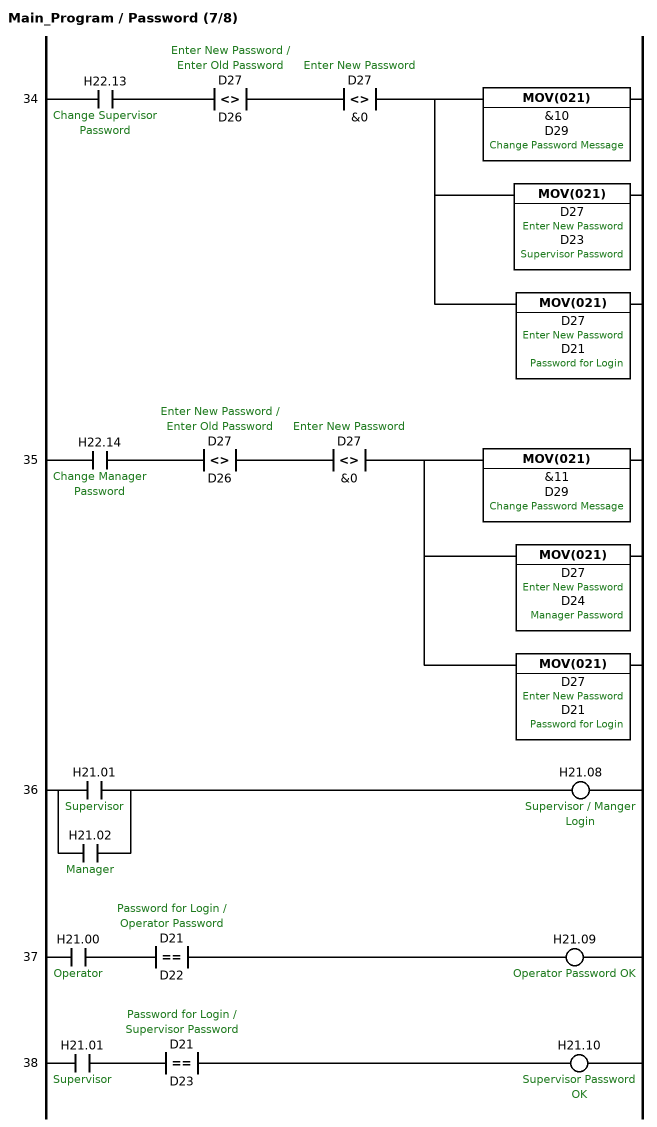
; rung 34
LD H22.13  ; Change Supervisor Password
AND<>(305) D27 D26  ; Enter New Password, Enter Old Password
AND<>(305) D27 &0  ; Enter New Password
MOV(021) &10 D29  ; Change Password Message
MOV(021) D27 D23  ; Enter New Password, Supervisor Password
MOV(021) D27 D21  ; Enter New Password, Password for Login
; rung 35
LD H22.14  ; Change Manager Password
AND<>(305) D27 D26  ; Enter New Password, Enter Old Password
AND<>(305) D27 &0  ; Enter New Password
MOV(021) &11 D29  ; Change Password Message
MOV(021) D27 D24  ; Enter New Password, Manager Password
MOV(021) D27 D21  ; Enter New Password, Password for Login
; rung 36
LD H21.01  ; Supervisor
OR H21.02  ; Manager
OUT H21.08  ; Supervisor / Manger Login
; rung 37
LD H21.00  ; Operator
AND=(300) D21 D22  ; Password for Login, Operator Password
OUT H21.09  ; Operator Password OK
; rung 38
LD H21.01  ; Supervisor
AND=(300) D21 D23  ; Password for Login, Supervisor Password
OUT H21.10  ; Supervisor Password OK

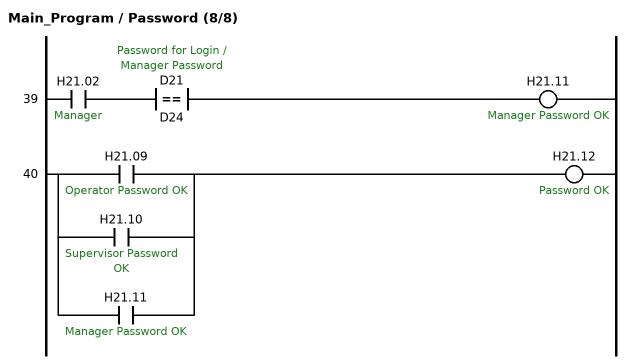
; rung 39
LD H21.02  ; Manager
AND=(300) D21 D24  ; Password for Login, Manager Password
OUT H21.11  ; Manager Password OK
; rung 40
LD H21.09  ; Operator Password OK
OR H21.10  ; Supervisor Password OK
OR H21.11  ; Manager Password OK
OUT H21.12  ; Password OK

### Section General

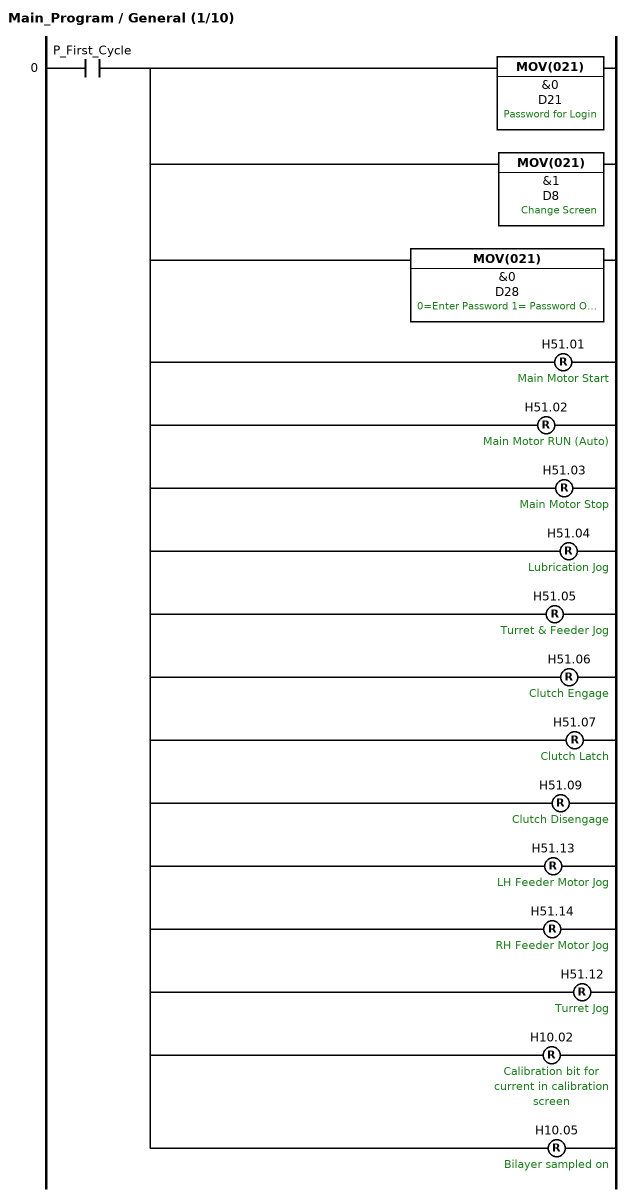
; rung 0
LD P_First_Cycle
MOV(021) &0 D21  ; Password for Login
MOV(021) &1 D8  ; Change Screen
MOV(021) &0 D28  ; 0=Enter Password 1= Password OK 2=Invalid Password
RSET H51.01  ; Main Motor Start
RSET H51.02  ; Main Motor RUN (Auto)
RSET H51.03  ; Main Motor Stop
RSET H51.04  ; Lubrication Jog
RSET H51.05  ; Turret & Feeder Jog
RSET H51.06  ; Clutch Engage
RSET H51.07  ; Clutch Latch
RSET H51.09  ; Clutch Disengage
RSET H51.13  ; LH Feeder Motor Jog
RSET H51.14  ; RH Feeder Motor Jog
RSET H51.12  ; Turret Jog
RSET H10.02  ; Calibration bit for current in calibration screen
RSET H10.05  ; Bilayer sampled on

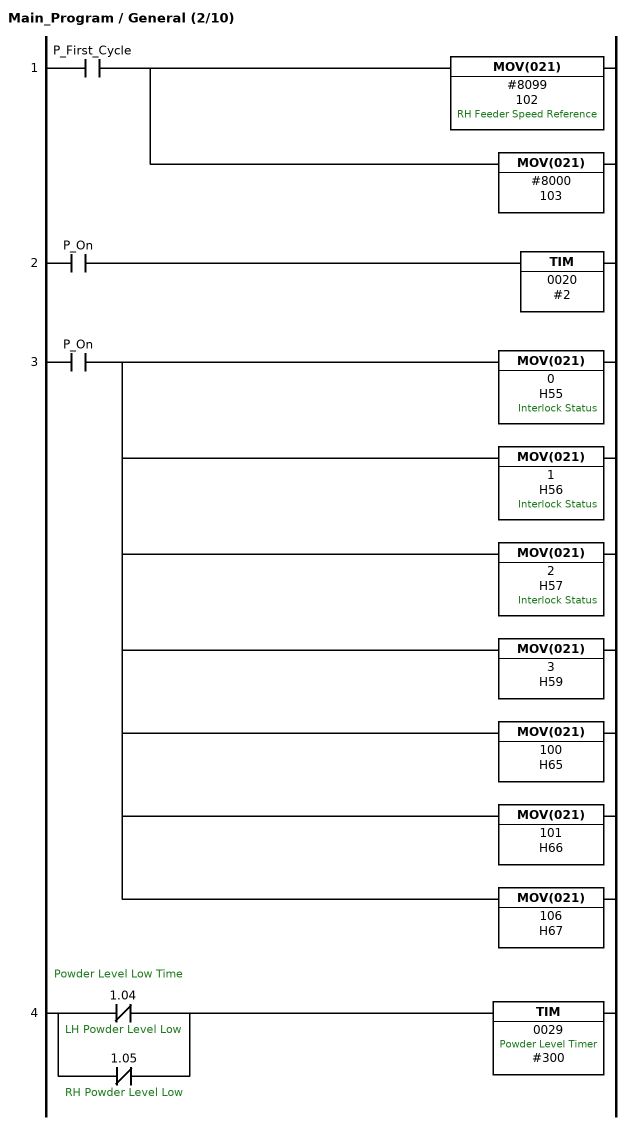
; rung 1
LD P_First_Cycle
MOV(021) #8099 102  ; RH Feeder Speed Reference
MOV(021) #8000 103
; rung 2
LD P_On
TIM 0020 #2
; rung 3
LD P_On
MOV(021) 0 H55  ; Interlock Status
MOV(021) 1 H56  ; Interlock Status
MOV(021) 2 H57  ; Interlock Status
MOV(021) 3 H59
MOV(021) 100 H65
MOV(021) 101 H66
MOV(021) 106 H67
; rung 4: Powder Level Low Time
LDNOT 1.04  ; LH Powder Level Low
ORNOT 1.05  ; RH Powder Level Low
TIM 0029 #300  ; Powder Level Timer

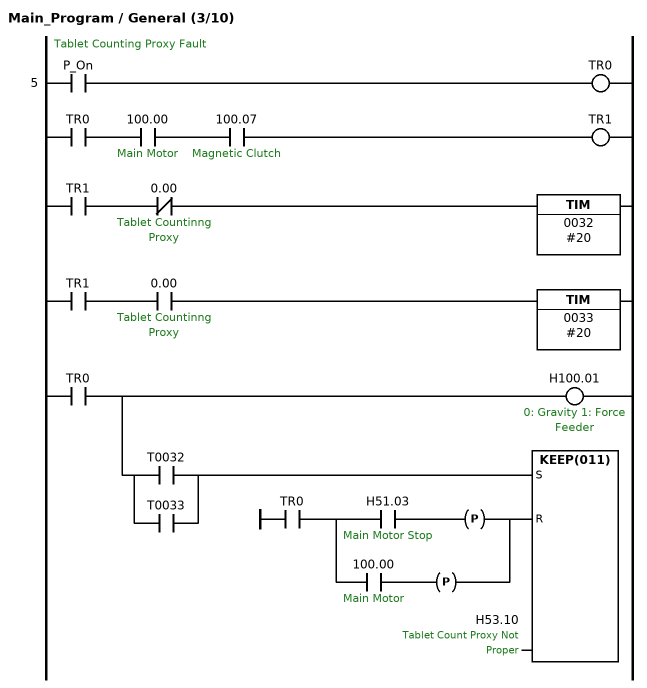
; rung 5: Tablet Counting Proxy Fault
LD P_On
OUT TR0
AND 100.00  ; Main Motor
AND 100.07  ; Magnetic Clutch
OUT TR1
ANDNOT 0.00  ; Tablet Countinng Proxy
TIM 0032 #20
LD TR1
AND 0.00  ; Tablet Countinng Proxy
TIM 0033 #20
LD TR0
OUT H100.01  ; 0: Gravity 1: Force Feeder
LD T0032
OR T0033
ANDLD
LD TR0
LD H51.03  ; Main Motor Stop
UP(521)
LD 100.00  ; Main Motor
UP(521)
ORLD
ANDLD
KEEP(011) H53.10  ; Tablet Count Proxy Not Proper

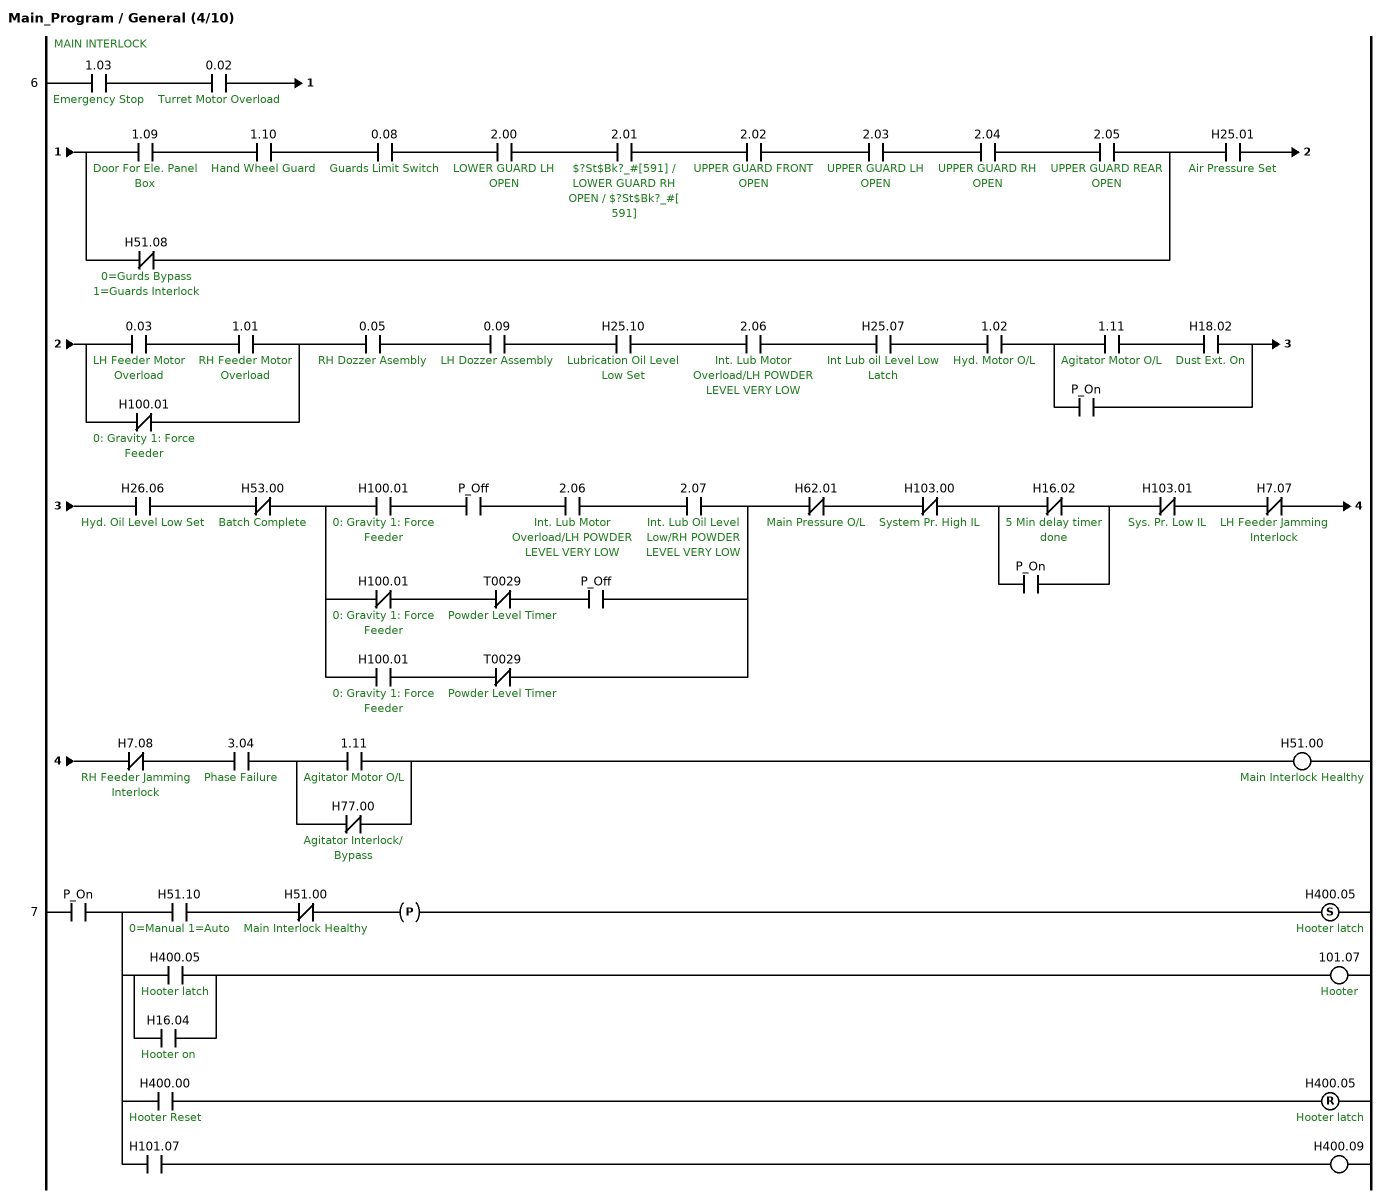
; rung 6: MAIN INTERLOCK
LD 1.03  ; Emergency Stop
AND 0.02  ; Turret Motor Overload
LD 1.09  ; Door For Ele. Panel Box
AND 1.10  ; Hand Wheel Guard
AND 0.08  ; Guards Limit Switch
AND 2.00  ; LOWER GUARD LH OPEN
AND 2.01  ; $?St$Bk?_#[591] / LOWER GUARD RH OPEN / $?St$Bk?_#[591]
AND 2.02  ; UPPER GUARD FRONT OPEN
AND 2.03  ; UPPER GUARD LH OPEN
AND 2.04  ; UPPER GUARD RH OPEN
AND 2.05  ; UPPER GUARD REAR OPEN
ORNOT H51.08  ; 0=Gurds Bypass 1=Guards Interlock
ANDLD
AND H25.01  ; Air Pressure Set
LD 0.03  ; LH Feeder Motor Overload
AND 1.01  ; RH Feeder Motor Overload
ORNOT H100.01  ; 0: Gravity 1: Force Feeder
ANDLD
AND 0.05  ; RH Dozzer Asembly
AND 0.09  ; LH Dozzer Assembly
AND H25.10  ; Lubrication Oil Level Low Set
AND 2.06  ; Int. Lub Motor Overload/LH POWDER LEVEL VERY LOW
AND H25.07  ; Int Lub oil Level Low Latch
AND 1.02  ; Hyd. Motor O/L
LD 1.11  ; Agitator Motor O/L
AND H18.02  ; Dust Ext. On
OR P_On
ANDLD
AND H26.06  ; Hyd. Oil Level Low Set
ANDNOT H53.00  ; Batch Complete
LD H100.01  ; 0: Gravity 1: Force Feeder
AND P_Off
AND 2.06  ; Int. Lub Motor Overload/LH POWDER LEVEL VERY LOW
AND 2.07  ; Int. Lub Oil Level Low/RH POWDER LEVEL VERY LOW
LDNOT H100.01  ; 0: Gravity 1: Force Feeder
ANDNOT T0029  ; Powder Level Timer
AND P_Off
ORLD
LD H100.01  ; 0: Gravity 1: Force Feeder
ANDNOT T0029  ; Powder Level Timer
ORLD
ANDLD
ANDNOT H62.01  ; Main Pressure O/L
ANDNOT H103.00  ; System Pr. High IL
LDNOT H16.02  ; 5 Min delay timer done
OR P_On
ANDLD
ANDNOT H103.01  ; Sys. Pr. Low IL
ANDNOT H7.07  ; LH Feeder Jamming Interlock
ANDNOT H7.08  ; RH Feeder Jamming Interlock
AND 3.04  ; Phase Failure
LD 1.11  ; Agitator Motor O/L
ORNOT H77.00  ; Agitator Interlock/Bypass
ANDLD
OUT H51.00  ; Main Interlock Healthy
; rung 7
LD P_On
OUT TR0
AND H51.10  ; 0=Manual 1=Auto
ANDNOT H51.00  ; Main Interlock Healthy
UP(521)
SET H400.05  ; Hooter latch
LD TR0
LD H400.05  ; Hooter latch
OR H16.04  ; Hooter on
ANDLD
OUT 101.07  ; Hooter
LD TR0
AND H400.00  ; Hooter Reset
RSET H400.05  ; Hooter latch
LD TR0
AND H101.07
OUT H400.09

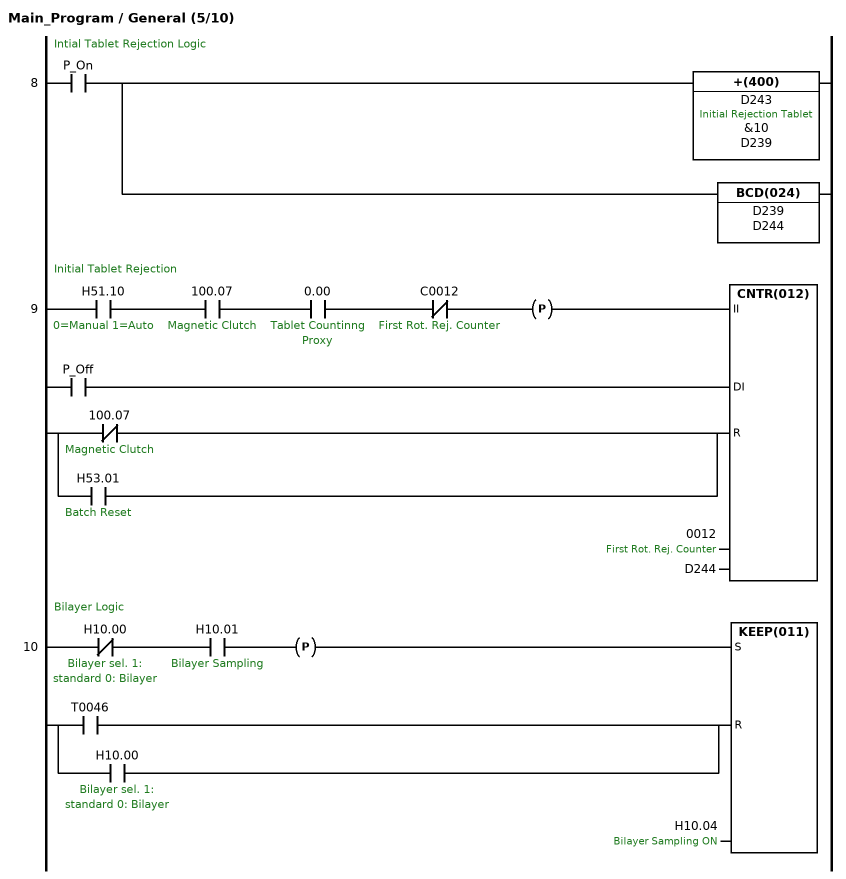
; rung 8: Intial Tablet Rejection Logic
LD P_On
+(400) D243 &10 D239  ; Initial Rejection Tablet
BCD(024) D239 D244
; rung 9: Initial Tablet Rejection
LD H51.10  ; 0=Manual 1=Auto
AND 100.07  ; Magnetic Clutch
AND 0.00  ; Tablet Countinng Proxy
ANDNOT C0012  ; First Rot. Rej. Counter
UP(521)
LD P_Off
LDNOT 100.07  ; Magnetic Clutch
OR H53.01  ; Batch Reset
CNTR(012) 0012 D244  ; First Rot. Rej. Counter
; rung 10: Bilayer Logic
LDNOT H10.00  ; Bilayer sel. 1: standard 0: Bilayer
AND H10.01  ; Bilayer Sampling
UP(521)
LD T0046
OR H10.00  ; Bilayer sel. 1: standard 0: Bilayer
KEEP(011) H10.04  ; Bilayer Sampling ON

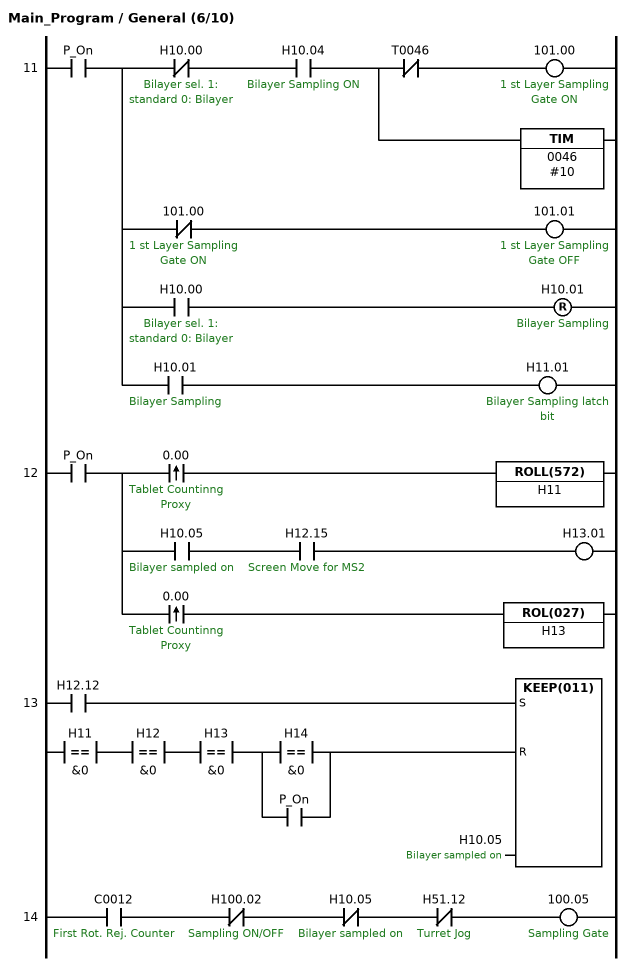
; rung 11
LD P_On
OUT TR0
ANDNOT H10.00  ; Bilayer sel. 1: standard 0: Bilayer
AND H10.04  ; Bilayer Sampling ON
OUT TR1
ANDNOT T0046
OUT 101.00  ; 1 st Layer Sampling Gate ON
LD TR1
TIM 0046 #10
LD TR0
ANDNOT 101.00  ; 1 st Layer Sampling Gate ON
OUT 101.01  ; 1 st Layer Sampling Gate OFF
LD TR0
AND H10.00  ; Bilayer sel. 1: standard 0: Bilayer
RSET H10.01  ; Bilayer Sampling
LD TR0
AND H10.01  ; Bilayer Sampling
OUT H11.01  ; Bilayer Sampling latch bit
; rung 12
LD P_On
OUT TR0
@AND 0.00  ; Tablet Countinng Proxy
ROLL(572) H11
LD TR0
AND H10.05  ; Bilayer sampled on
AND H12.15  ; Screen Move for MS2
OUT H13.01
LD TR0
@AND 0.00  ; Tablet Countinng Proxy
ROL(027) H13
; rung 13
LD H12.12
LD=(300) H11 &0
AND=(300) H12 &0
AND=(300) H13 &0
LD=(300) H14 &0
OR P_On
ANDLD
KEEP(011) H10.05  ; Bilayer sampled on
; rung 14
LD C0012  ; First Rot. Rej. Counter
ANDNOT H100.02  ; Sampling ON/OFF
ANDNOT H10.05  ; Bilayer sampled on
ANDNOT H51.12  ; Turret Jog
OUT 100.05  ; Sampling Gate

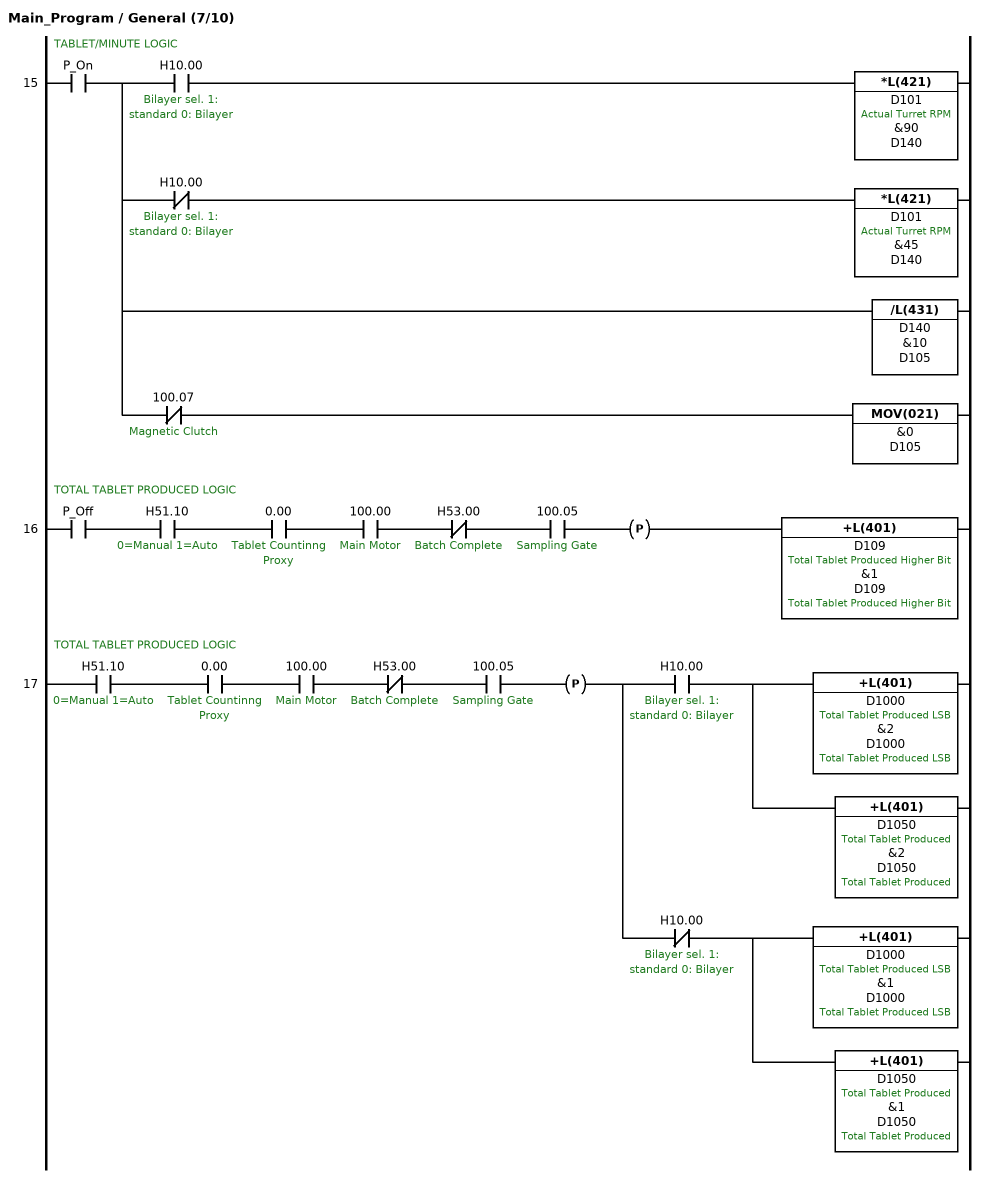
; rung 15: TABLET/MINUTE LOGIC
LD P_On
OUT TR0
AND H10.00  ; Bilayer sel. 1: standard 0: Bilayer
*L(421) D101 &90 D140  ; Actual Turret RPM
LD TR0
ANDNOT H10.00  ; Bilayer sel. 1: standard 0: Bilayer
*L(421) D101 &45 D140  ; Actual Turret RPM
LD TR0
/L(431) D140 &10 D105
ANDNOT 100.07  ; Magnetic Clutch
MOV(021) &0 D105
; rung 16: TOTAL TABLET PRODUCED LOGIC
LD P_Off
AND H51.10  ; 0=Manual 1=Auto
AND 0.00  ; Tablet Countinng Proxy
AND 100.00  ; Main Motor
ANDNOT H53.00  ; Batch Complete
AND 100.05  ; Sampling Gate
UP(521)
+L(401) D109 &1 D109  ; Total Tablet Produced Higher Bit
; rung 17: TOTAL TABLET PRODUCED LOGIC
LD H51.10  ; 0=Manual 1=Auto
AND 0.00  ; Tablet Countinng Proxy
AND 100.00  ; Main Motor
ANDNOT H53.00  ; Batch Complete
AND 100.05  ; Sampling Gate
UP(521)
OUT TR0
AND H10.00  ; Bilayer sel. 1: standard 0: Bilayer
+L(401) D1000 &2 D1000  ; Total Tablet Produced LSB
+L(401) D1050 &2 D1050  ; Total Tablet Produced
LD TR0
ANDNOT H10.00  ; Bilayer sel. 1: standard 0: Bilayer
+L(401) D1000 &1 D1000  ; Total Tablet Produced LSB
+L(401) D1050 &1 D1050  ; Total Tablet Produced

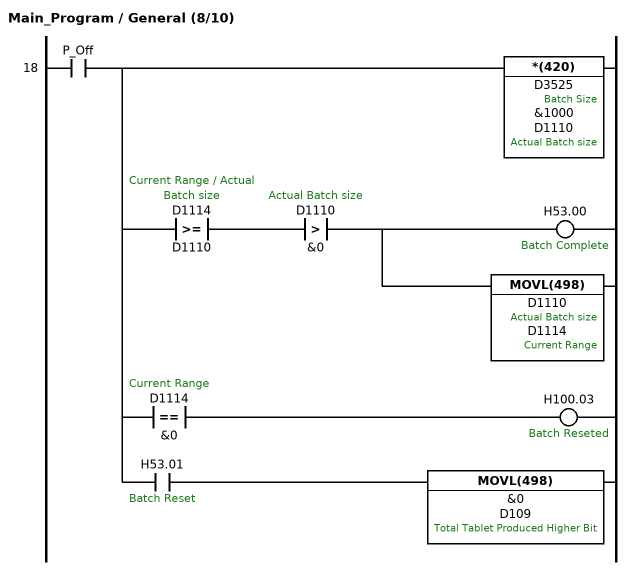
; rung 18
LD P_Off
OUT TR0
*(420) D3525 &1000 D1110  ; Batch Size, Actual Batch size
AND>=L(326) D1114 D1110  ; Current Range, Actual Batch size
AND>L(321) D1110 &0  ; Actual Batch size
OUT H53.00  ; Batch Complete
MOVL(498) D1110 D1114  ; Actual Batch size, Current Range
LD TR0
AND=L(301) D1114 &0  ; Current Range
OUT H100.03  ; Batch Reseted
LD TR0
AND H53.01  ; Batch Reset
MOVL(498) &0 D109  ; Total Tablet Produced Higher Bit

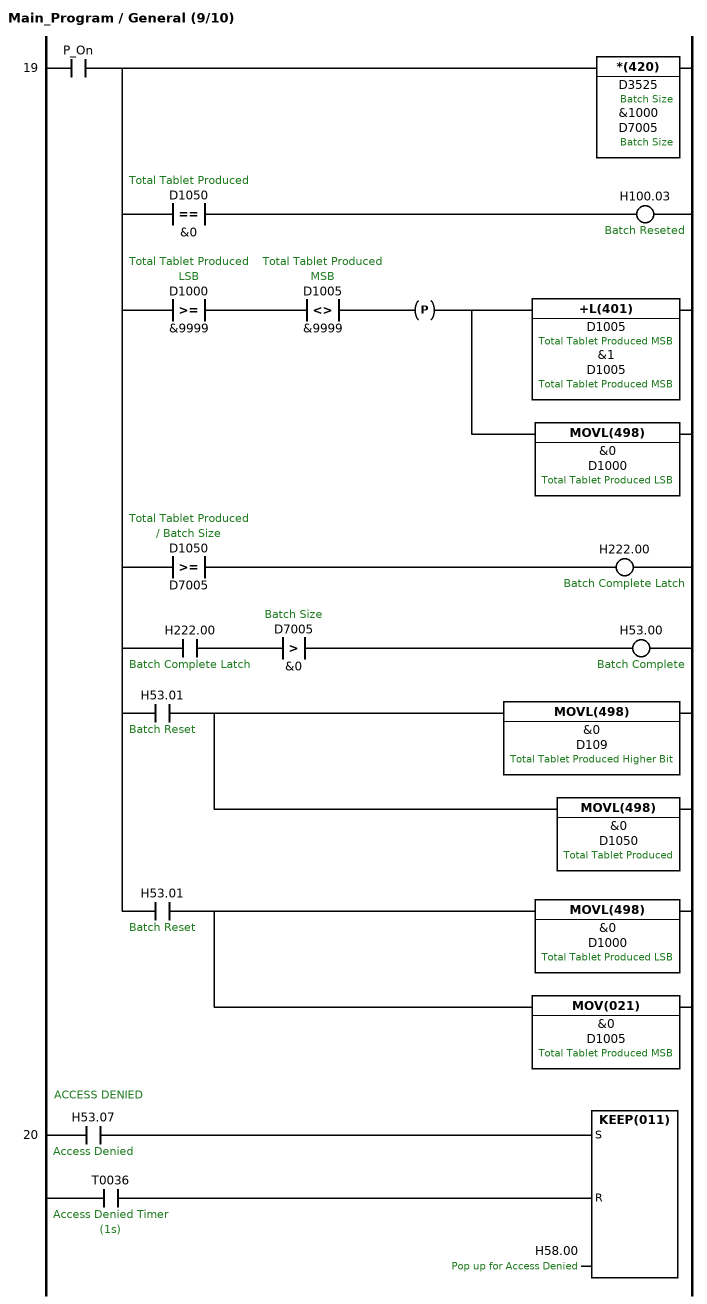
; rung 19
LD P_On
OUT TR0
*(420) D3525 &1000 D7005  ; Batch Size
AND=L(301) D1050 &0  ; Total Tablet Produced
OUT H100.03  ; Batch Reseted
LD TR0
AND>=(325) D1000 &9999  ; Total Tablet Produced LSB
AND<>(305) D1005 &9999  ; Total Tablet Produced MSB
UP(521)
+L(401) D1005 &1 D1005  ; Total Tablet Produced MSB
MOVL(498) &0 D1000  ; Total Tablet Produced LSB
LD TR0
AND>=L(326) D1050 D7005  ; Total Tablet Produced, Batch Size
OUT H222.00  ; Batch Complete Latch
LD TR0
AND H222.00  ; Batch Complete Latch
AND>L(321) D7005 &0  ; Batch Size
OUT H53.00  ; Batch Complete
LD TR0
AND H53.01  ; Batch Reset
MOVL(498) &0 D109  ; Total Tablet Produced Higher Bit
MOVL(498) &0 D1050  ; Total Tablet Produced
LD TR0
AND H53.01  ; Batch Reset
MOVL(498) &0 D1000  ; Total Tablet Produced LSB
MOV(021) &0 D1005  ; Total Tablet Produced MSB
; rung 20: ACCESS DENIED
LD H53.07  ; Access Denied
LD T0036  ; Access Denied Timer (1s)
KEEP(011) H58.00  ; Pop up for Access Denied

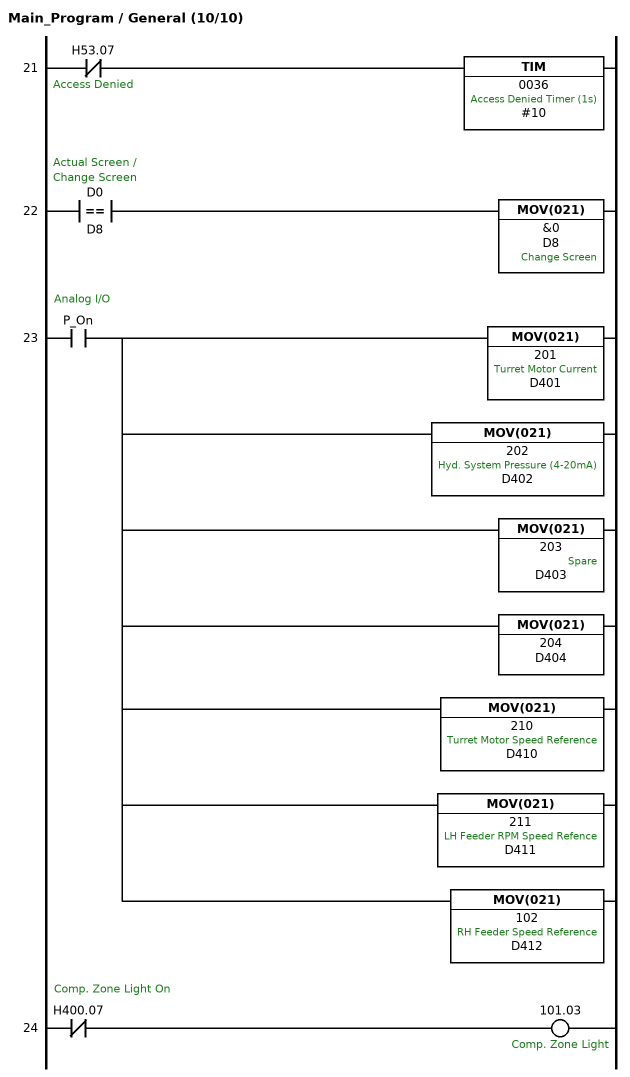
; rung 21
LDNOT H53.07  ; Access Denied
TIM 0036 #10  ; Access Denied Timer (1s)
; rung 22
LD=(300) D0 D8  ; Actual Screen, Change Screen
MOV(021) &0 D8  ; Change Screen
; rung 23: Analog I/O
LD P_On
MOV(021) 201 D401  ; Turret Motor Current
MOV(021) 202 D402  ; Hyd. System Pressure (4-20mA)
MOV(021) 203 D403  ; Spare
MOV(021) 204 D404
MOV(021) 210 D410  ; Turret Motor Speed Reference
MOV(021) 211 D411  ; LH Feeder RPM Speed Refence
MOV(021) 102 D412  ; RH Feeder Speed Reference
; rung 24: Comp. Zone Light On
LDNOT H400.07
OUT 101.03  ; Comp. Zone Light

### Section Turret_feeder

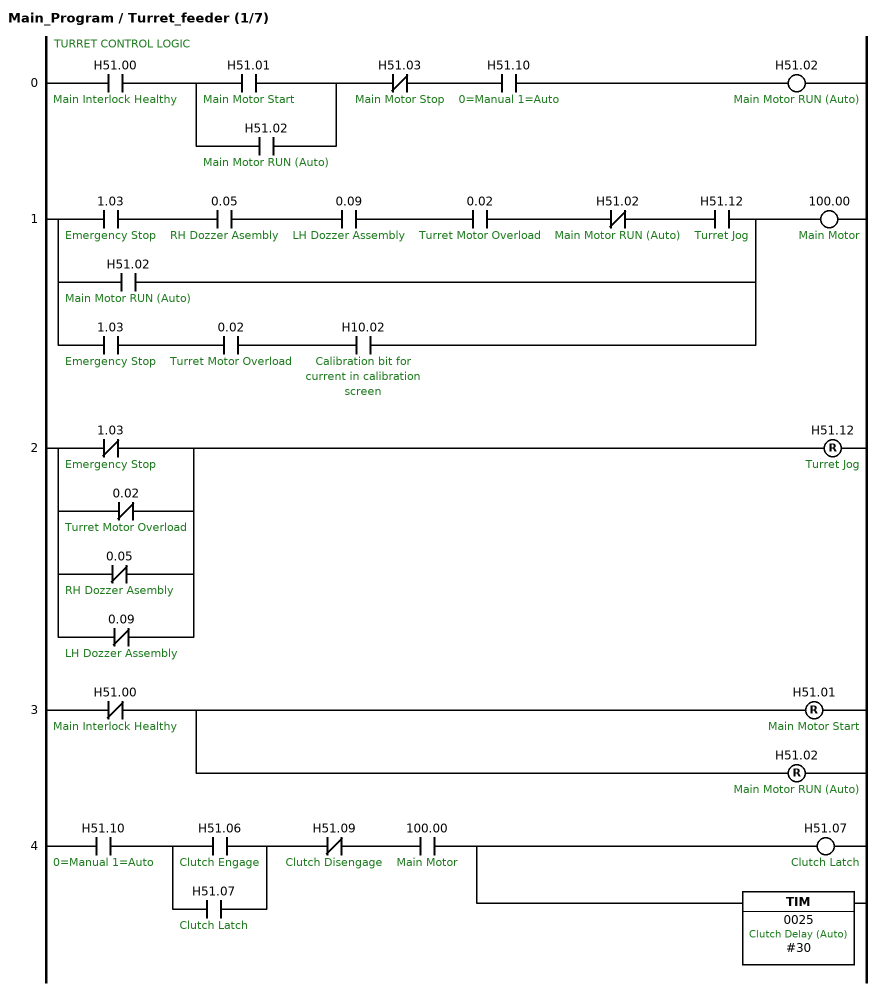
; rung 0: TURRET CONTROL LOGIC
LD H51.00  ; Main Interlock Healthy
LD H51.01  ; Main Motor Start
OR H51.02  ; Main Motor RUN (Auto)
ANDLD
ANDNOT H51.03  ; Main Motor Stop
AND H51.10  ; 0=Manual 1=Auto
OUT H51.02  ; Main Motor RUN (Auto)
; rung 1
LD 1.03  ; Emergency Stop
AND 0.05  ; RH Dozzer Asembly
AND 0.09  ; LH Dozzer Assembly
AND 0.02  ; Turret Motor Overload
ANDNOT H51.02  ; Main Motor RUN (Auto)
AND H51.12  ; Turret Jog
OR H51.02  ; Main Motor RUN (Auto)
LD 1.03  ; Emergency Stop
AND 0.02  ; Turret Motor Overload
AND H10.02  ; Calibration bit for current in calibration screen
ORLD
OUT 100.00  ; Main Motor
; rung 2
LDNOT 1.03  ; Emergency Stop
ORNOT 0.02  ; Turret Motor Overload
ORNOT 0.05  ; RH Dozzer Asembly
ORNOT 0.09  ; LH Dozzer Assembly
RSET H51.12  ; Turret Jog
; rung 3
LDNOT H51.00  ; Main Interlock Healthy
RSET H51.01  ; Main Motor Start
RSET H51.02  ; Main Motor RUN (Auto)
; rung 4
LD H51.10  ; 0=Manual 1=Auto
LD H51.06  ; Clutch Engage
OR H51.07  ; Clutch Latch
ANDLD
ANDNOT H51.09  ; Clutch Disengage
AND 100.00  ; Main Motor
OUT H51.07  ; Clutch Latch
TIM 0025 #30  ; Clutch Delay (Auto)

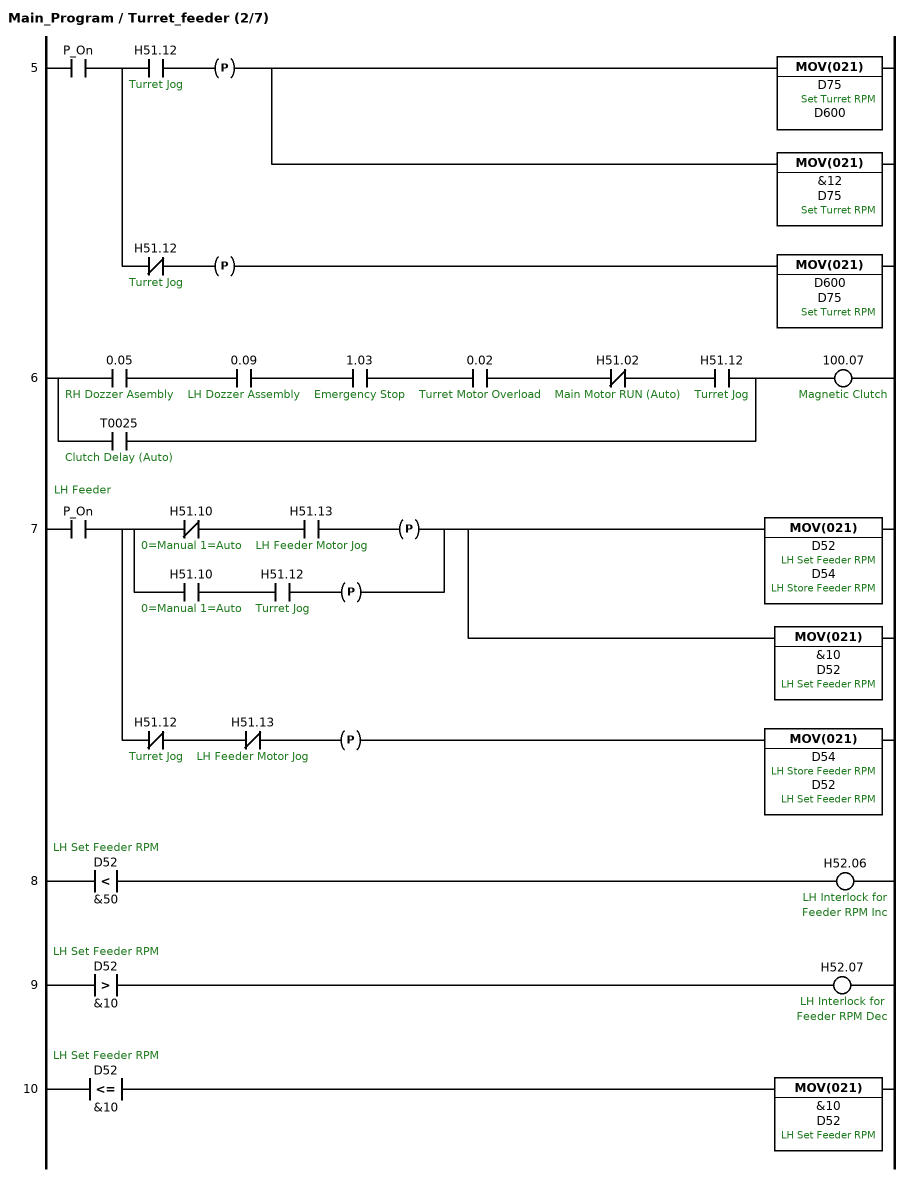
; rung 5
LD P_On
OUT TR0
AND H51.12  ; Turret Jog
UP(521)
MOV(021) D75 D600  ; Set Turret RPM
MOV(021) &12 D75  ; Set Turret RPM
LD TR0
ANDNOT H51.12  ; Turret Jog
UP(521)
MOV(021) D600 D75  ; Set Turret RPM
; rung 6
LD 0.05  ; RH Dozzer Asembly
AND 0.09  ; LH Dozzer Assembly
AND 1.03  ; Emergency Stop
AND 0.02  ; Turret Motor Overload
ANDNOT H51.02  ; Main Motor RUN (Auto)
AND H51.12  ; Turret Jog
OR T0025  ; Clutch Delay (Auto)
OUT 100.07  ; Magnetic Clutch
; rung 7: LH Feeder
LD P_On
OUT TR0
LDNOT H51.10  ; 0=Manual 1=Auto
AND H51.13  ; LH Feeder Motor Jog
UP(521)
LD H51.10  ; 0=Manual 1=Auto
AND H51.12  ; Turret Jog
UP(521)
ORLD
ANDLD
MOV(021) D52 D54  ; LH Set Feeder RPM, LH Store Feeder RPM
MOV(021) &10 D52  ; LH Set Feeder RPM
LD TR0
ANDNOT H51.12  ; Turret Jog
ANDNOT H51.13  ; LH Feeder Motor Jog
UP(521)
MOV(021) D54 D52  ; LH Store Feeder RPM, LH Set Feeder RPM
; rung 8
LD<(310) D52 &50  ; LH Set Feeder RPM
OUT H52.06  ; LH Interlock for Feeder RPM Inc
; rung 9
LD>(320) D52 &10  ; LH Set Feeder RPM
OUT H52.07  ; LH Interlock for Feeder RPM Dec
; rung 10
LD<=(315) D52 &10  ; LH Set Feeder RPM
MOV(021) &10 D52  ; LH Set Feeder RPM

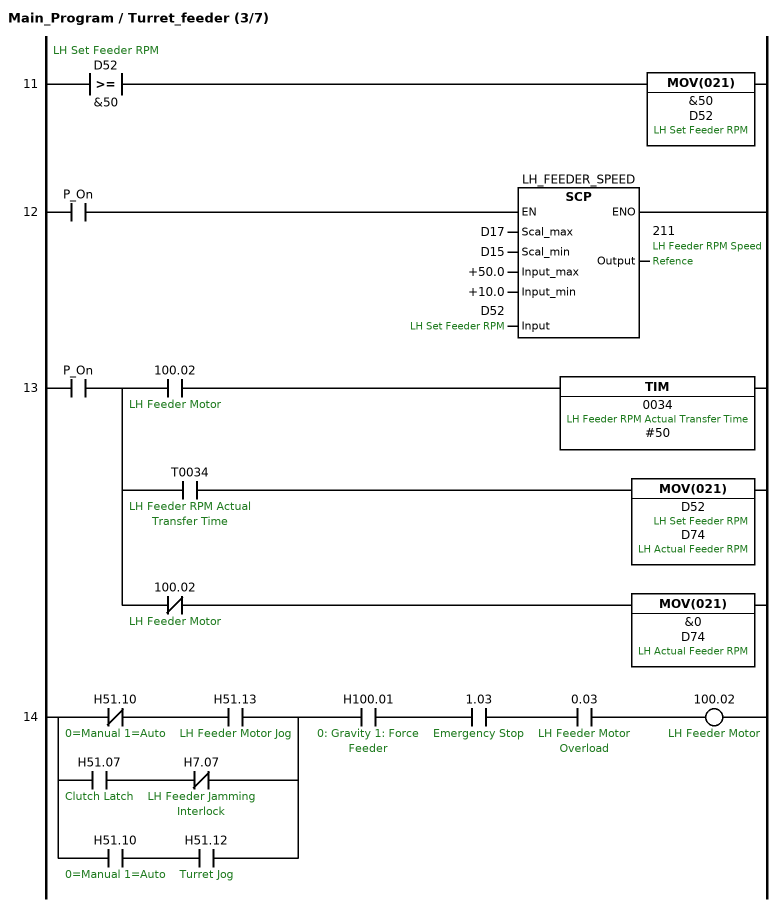
; rung 11
LD>=(325) D52 &50  ; LH Set Feeder RPM
MOV(021) &50 D52  ; LH Set Feeder RPM
; rung 12
LD P_On
CALL LH_FEEDER_SPEED : SCP (Scal_max := D17, Scal_min := D15, Input_max := +50.0, Input_min := +10.0, Input := D52, Output => 211)  ; LH Set Feeder RPM, LH Feeder RPM Speed Refence
; rung 13
LD P_On
OUT TR0
AND 100.02  ; LH Feeder Motor
TIM 0034 #50  ; LH Feeder RPM Actual Transfer Time
LD TR0
AND T0034  ; LH Feeder RPM Actual Transfer Time
MOV(021) D52 D74  ; LH Set Feeder RPM, LH Actual Feeder RPM
LD TR0
ANDNOT 100.02  ; LH Feeder Motor
MOV(021) &0 D74  ; LH Actual Feeder RPM
; rung 14
LDNOT H51.10  ; 0=Manual 1=Auto
AND H51.13  ; LH Feeder Motor Jog
LD H51.07  ; Clutch Latch
ANDNOT H7.07  ; LH Feeder Jamming Interlock
ORLD
LD H51.10  ; 0=Manual 1=Auto
AND H51.12  ; Turret Jog
ORLD
AND H100.01  ; 0: Gravity 1: Force Feeder
AND 1.03  ; Emergency Stop
AND 0.03  ; LH Feeder Motor Overload
OUT 100.02  ; LH Feeder Motor

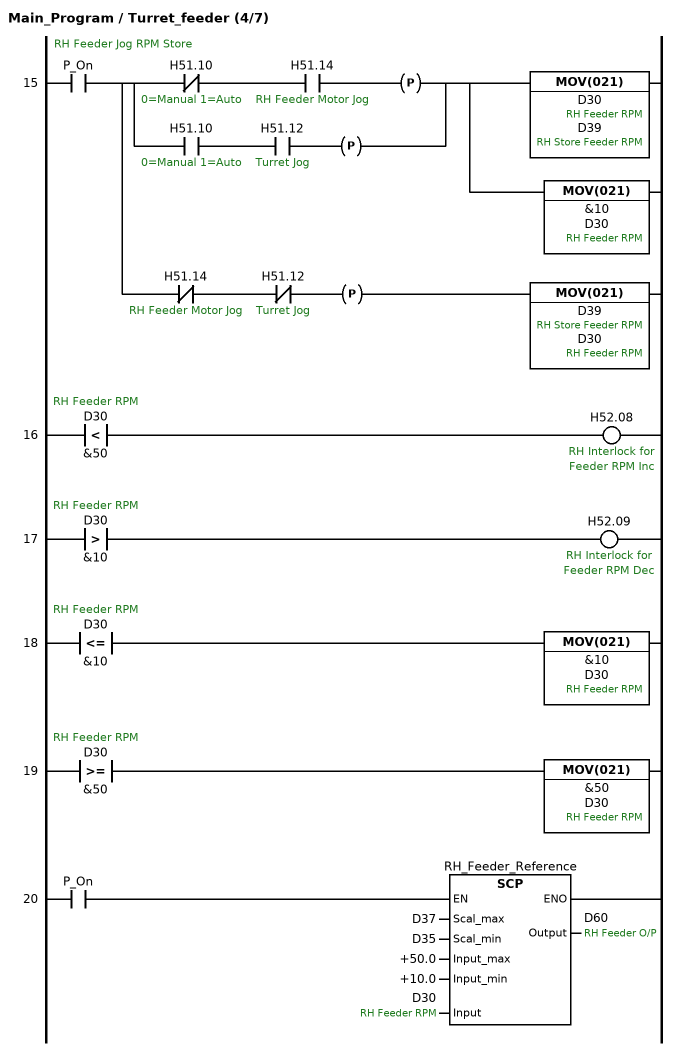
; rung 15: RH Feeder Jog RPM Store
LD P_On
OUT TR0
LDNOT H51.10  ; 0=Manual 1=Auto
AND H51.14  ; RH Feeder Motor Jog
UP(521)
LD H51.10  ; 0=Manual 1=Auto
AND H51.12  ; Turret Jog
UP(521)
ORLD
ANDLD
MOV(021) D30 D39  ; RH Feeder RPM, RH Store Feeder RPM
MOV(021) &10 D30  ; RH Feeder RPM
LD TR0
ANDNOT H51.14  ; RH Feeder Motor Jog
ANDNOT H51.12  ; Turret Jog
UP(521)
MOV(021) D39 D30  ; RH Store Feeder RPM, RH Feeder RPM
; rung 16
LD<(310) D30 &50  ; RH Feeder RPM
OUT H52.08  ; RH Interlock for Feeder RPM Inc
; rung 17
LD>(320) D30 &10  ; RH Feeder RPM
OUT H52.09  ; RH Interlock for Feeder RPM Dec
; rung 18
LD<=(315) D30 &10  ; RH Feeder RPM
MOV(021) &10 D30  ; RH Feeder RPM
; rung 19
LD>=(325) D30 &50  ; RH Feeder RPM
MOV(021) &50 D30  ; RH Feeder RPM
; rung 20
LD P_On
CALL RH_Feeder_Reference : SCP (Scal_max := D37, Scal_min := D35, Input_max := +50.0, Input_min := +10.0, Input := D30, Output => D60)  ; RH Feeder RPM, RH Feeder O/P

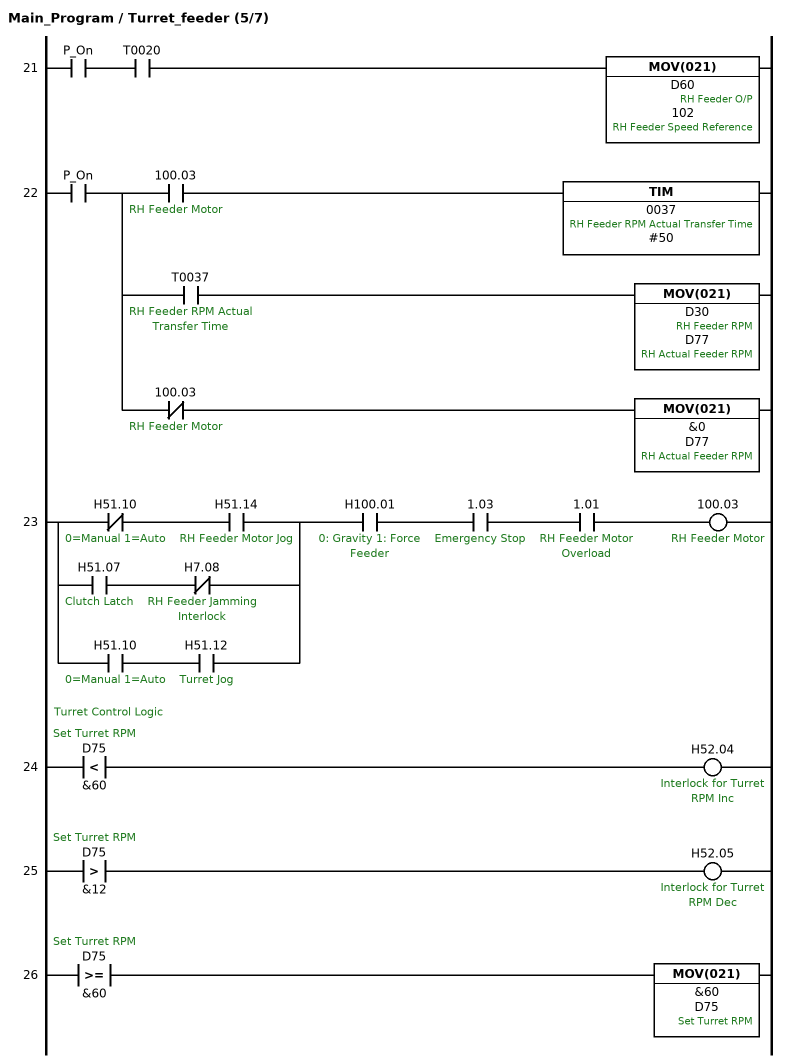
; rung 21
LD P_On
AND T0020
MOV(021) D60 102  ; RH Feeder O/P, RH Feeder Speed Reference
; rung 22
LD P_On
OUT TR0
AND 100.03  ; RH Feeder Motor
TIM 0037 #50  ; RH Feeder RPM Actual Transfer Time
LD TR0
AND T0037  ; RH Feeder RPM Actual Transfer Time
MOV(021) D30 D77  ; RH Feeder RPM, RH Actual Feeder RPM
LD TR0
ANDNOT 100.03  ; RH Feeder Motor
MOV(021) &0 D77  ; RH Actual Feeder RPM
; rung 23
LDNOT H51.10  ; 0=Manual 1=Auto
AND H51.14  ; RH Feeder Motor Jog
LD H51.07  ; Clutch Latch
ANDNOT H7.08  ; RH Feeder Jamming Interlock
ORLD
LD H51.10  ; 0=Manual 1=Auto
AND H51.12  ; Turret Jog
ORLD
AND H100.01  ; 0: Gravity 1: Force Feeder
AND 1.03  ; Emergency Stop
AND 1.01  ; RH Feeder Motor Overload
OUT 100.03  ; RH Feeder Motor
; rung 24: Turret Control Logic
LD<(310) D75 &60  ; Set Turret RPM
OUT H52.04  ; Interlock for Turret RPM Inc
; rung 25
LD>(320) D75 &12  ; Set Turret RPM
OUT H52.05  ; Interlock for Turret RPM Dec
; rung 26
LD>=(325) D75 &60  ; Set Turret RPM
MOV(021) &60 D75  ; Set Turret RPM

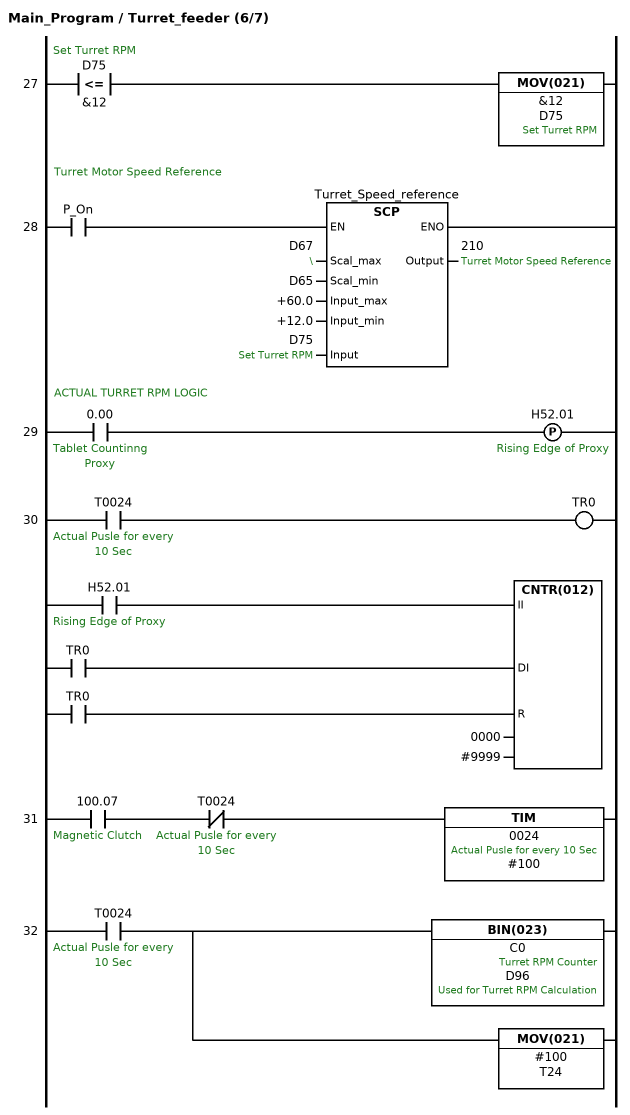
; rung 27
LD<=(315) D75 &12  ; Set Turret RPM
MOV(021) &12 D75  ; Set Turret RPM
; rung 28: Turret Motor Speed Reference
LD P_On
CALL Turret_Speed_reference : SCP (Scal_max := D67, Scal_min := D65, Input_max := +60.0, Input_min := +12.0, Input := D75, Output => 210)  ; \, Set Turret RPM, Turret Motor Speed Reference
; rung 29: ACTUAL TURRET RPM LOGIC
LD 0.00  ; Tablet Countinng Proxy
DIFU(013) H52.01  ; Rising Edge of Proxy
; rung 30
LD H52.01  ; Rising Edge of Proxy
LD T0024  ; Actual Pusle for every 10 Sec
OUT TR0
LD TR0
CNTR(012) 0000 #9999
; rung 31
LD 100.07  ; Magnetic Clutch
ANDNOT T0024  ; Actual Pusle for every 10 Sec
TIM 0024 #100  ; Actual Pusle for every 10 Sec
; rung 32
LD T0024  ; Actual Pusle for every 10 Sec
BIN(023) C0 D96  ; Turret RPM Counter, Used for Turret RPM Calculation
MOV(021) #100 T24

